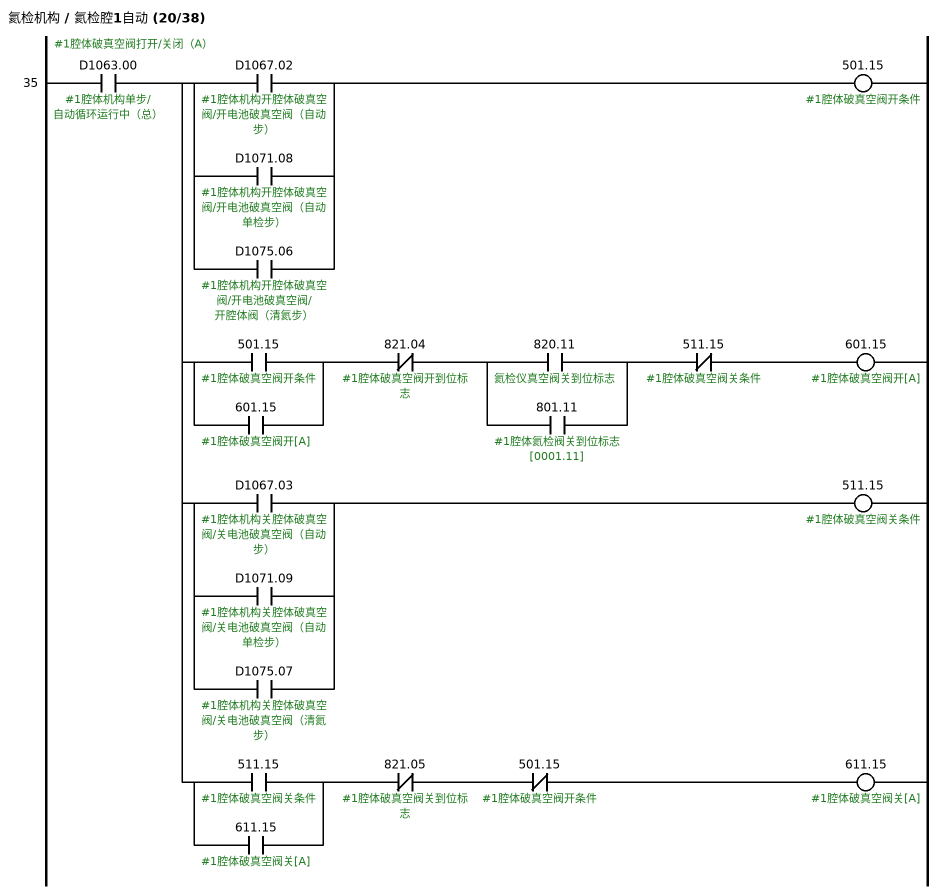
; [picture p216: 氦检机构 / 氦检腔1自动, rungs 35-35]
; rung 35: #1腔体破真空阀打开/关闭（A）
LD D1063.00  ; #1腔体机构单步/自动循环运行中（总）
OUT TR0
LD D1067.02  ; #1腔体机构开腔体破真空阀/开电池破真空阀（自动步）
OR D1071.08  ; #1腔体机构开腔体破真空阀/开电池破真空阀（自动单检步）
OR D1075.06  ; #1腔体机构开腔体破真空阀/开电池破真空阀/开腔体阀（清氦步）
ANDLD
OUT 501.15  ; #1腔体破真空阀开条件
LD TR0
LD 501.15  ; #1腔体破真空阀开条件
OR 601.15  ; #1腔体破真空阀开[A]
ANDLD
ANDNOT 821.04  ; #1腔体破真空阀开到位标志
LD 820.11  ; 氦检仪真空阀关到位标志
OR 801.11  ; #1腔体氦检阀关到位标志[0001.11]
ANDLD
ANDNOT 511.15  ; #1腔体破真空阀关条件
OUT 601.15  ; #1腔体破真空阀开[A]
LD TR0
LD D1067.03  ; #1腔体机构关腔体破真空阀/关电池破真空阀（自动步）
OR D1071.09  ; #1腔体机构关腔体破真空阀/关电池破真空阀（自动单检步）
OR D1075.07  ; #1腔体机构关腔体破真空阀/关电池破真空阀（清氦步）
ANDLD
OUT 511.15  ; #1腔体破真空阀关条件
LD TR0
LD 511.15  ; #1腔体破真空阀关条件
OR 611.15  ; #1腔体破真空阀关[A]
ANDLD
ANDNOT 821.05  ; #1腔体破真空阀关到位标志
ANDNOT 501.15  ; #1腔体破真空阀开条件
OUT 611.15  ; #1腔体破真空阀关[A]

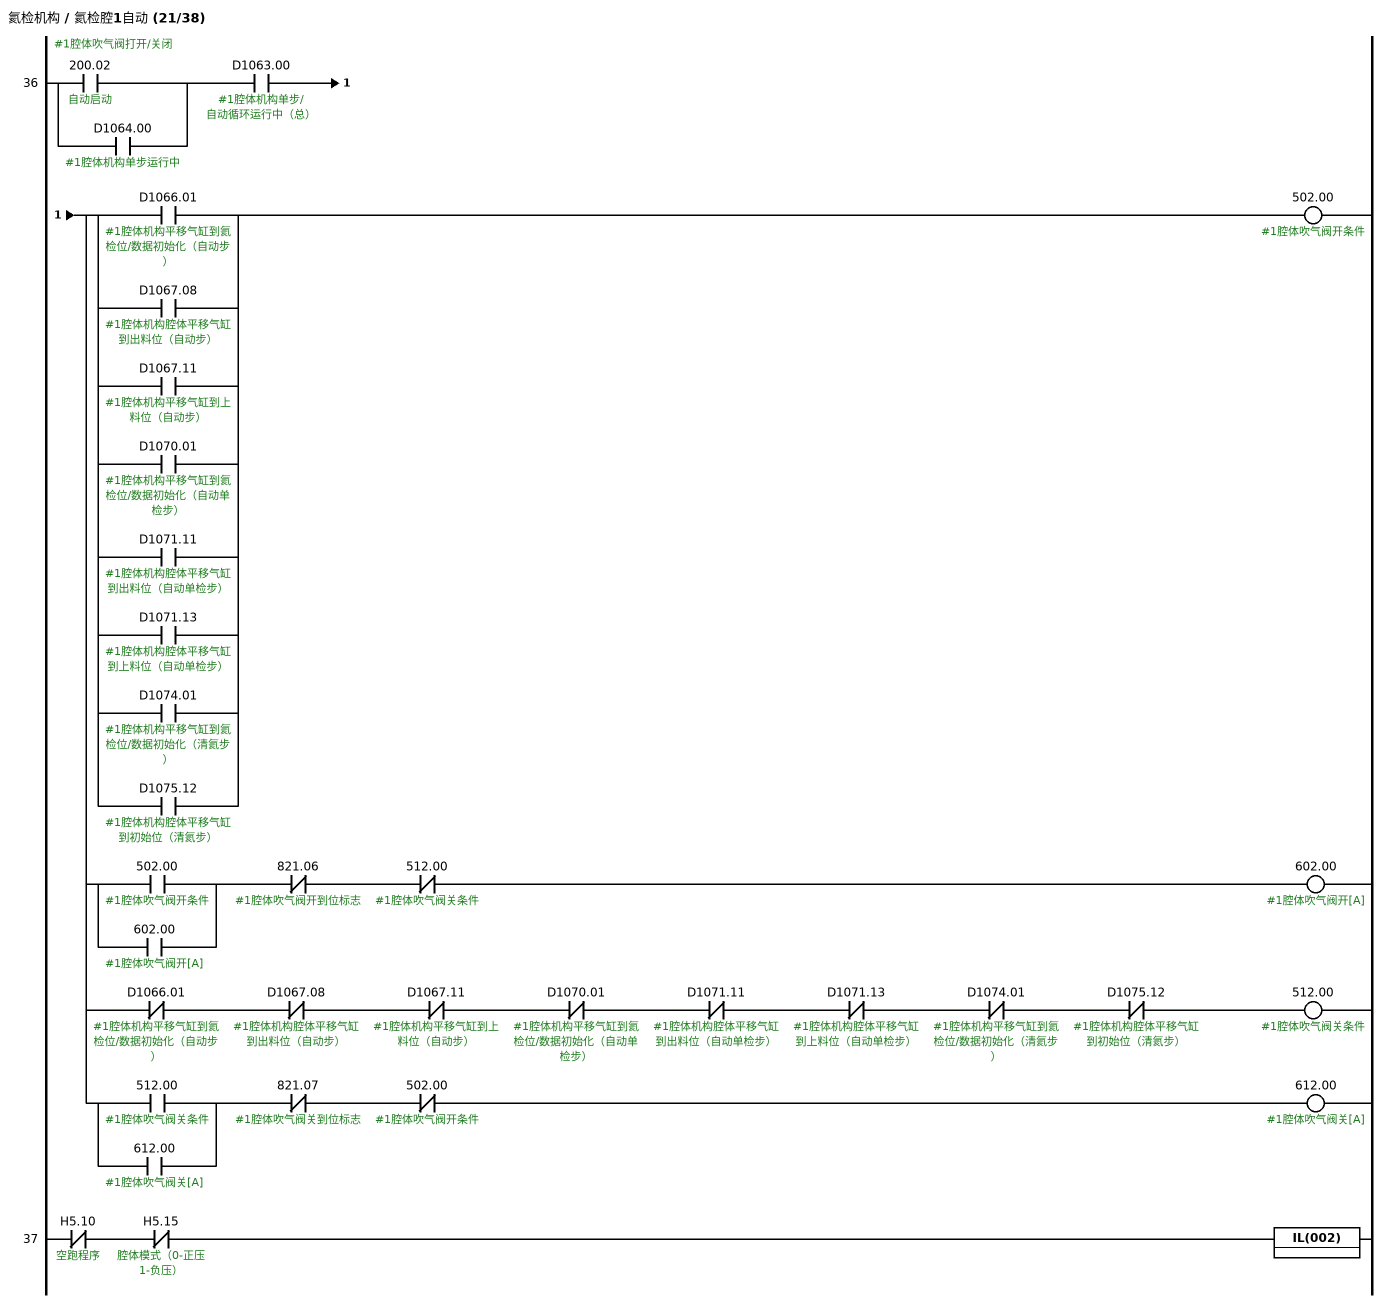
; rung 36: #1腔体吹气阀打开/关闭
LD 200.02  ; 自动启动
OR D1064.00  ; #1腔体机构单步运行中
AND D1063.00  ; #1腔体机构单步/自动循环运行中（总）
OUT TR0
LD D1066.01  ; #1腔体机构平移气缸到氦检位/数据初始化（自动步）
OR D1067.08  ; #1腔体机构腔体平移气缸到出料位（自动步）
OR D1067.11  ; #1腔体机构平移气缸到上料位（自动步）
OR D1070.01  ; #1腔体机构平移气缸到氦检位/数据初始化（自动单检步）
OR D1071.11  ; #1腔体机构腔体平移气缸到出料位（自动单检步）
OR D1071.13  ; #1腔体机构腔体平移气缸到上料位（自动单检步）
OR D1074.01  ; #1腔体机构平移气缸到氦检位/数据初始化（清氦步）
OR D1075.12  ; #1腔体机构腔体平移气缸到初始位（清氦步）
ANDLD
OUT 502.00  ; #1腔体吹气阀开条件
LD TR0
LD 502.00  ; #1腔体吹气阀开条件
OR 602.00  ; #1腔体吹气阀开[A]
ANDLD
ANDNOT 821.06  ; #1腔体吹气阀开到位标志
ANDNOT 512.00  ; #1腔体吹气阀关条件
OUT 602.00  ; #1腔体吹气阀开[A]
LD TR0
ANDNOT D1066.01  ; #1腔体机构平移气缸到氦检位/数据初始化（自动步）
ANDNOT D1067.08  ; #1腔体机构腔体平移气缸到出料位（自动步）
ANDNOT D1067.11  ; #1腔体机构平移气缸到上料位（自动步）
ANDNOT D1070.01  ; #1腔体机构平移气缸到氦检位/数据初始化（自动单检步）
ANDNOT D1071.11  ; #1腔体机构腔体平移气缸到出料位（自动单检步）
ANDNOT D1071.13  ; #1腔体机构腔体平移气缸到上料位（自动单检步）
ANDNOT D1074.01  ; #1腔体机构平移气缸到氦检位/数据初始化（清氦步）
ANDNOT D1075.12  ; #1腔体机构腔体平移气缸到初始位（清氦步）
OUT 512.00  ; #1腔体吹气阀关条件
LD TR0
LD 512.00  ; #1腔体吹气阀关条件
OR 612.00  ; #1腔体吹气阀关[A]
ANDLD
ANDNOT 821.07  ; #1腔体吹气阀关到位标志
ANDNOT 502.00  ; #1腔体吹气阀开条件
OUT 612.00  ; #1腔体吹气阀关[A]
; rung 37
LDNOT H5.10  ; 空跑程序
ANDNOT H5.15  ; 腔体模式（0-正压 1-负压）
IL(002)

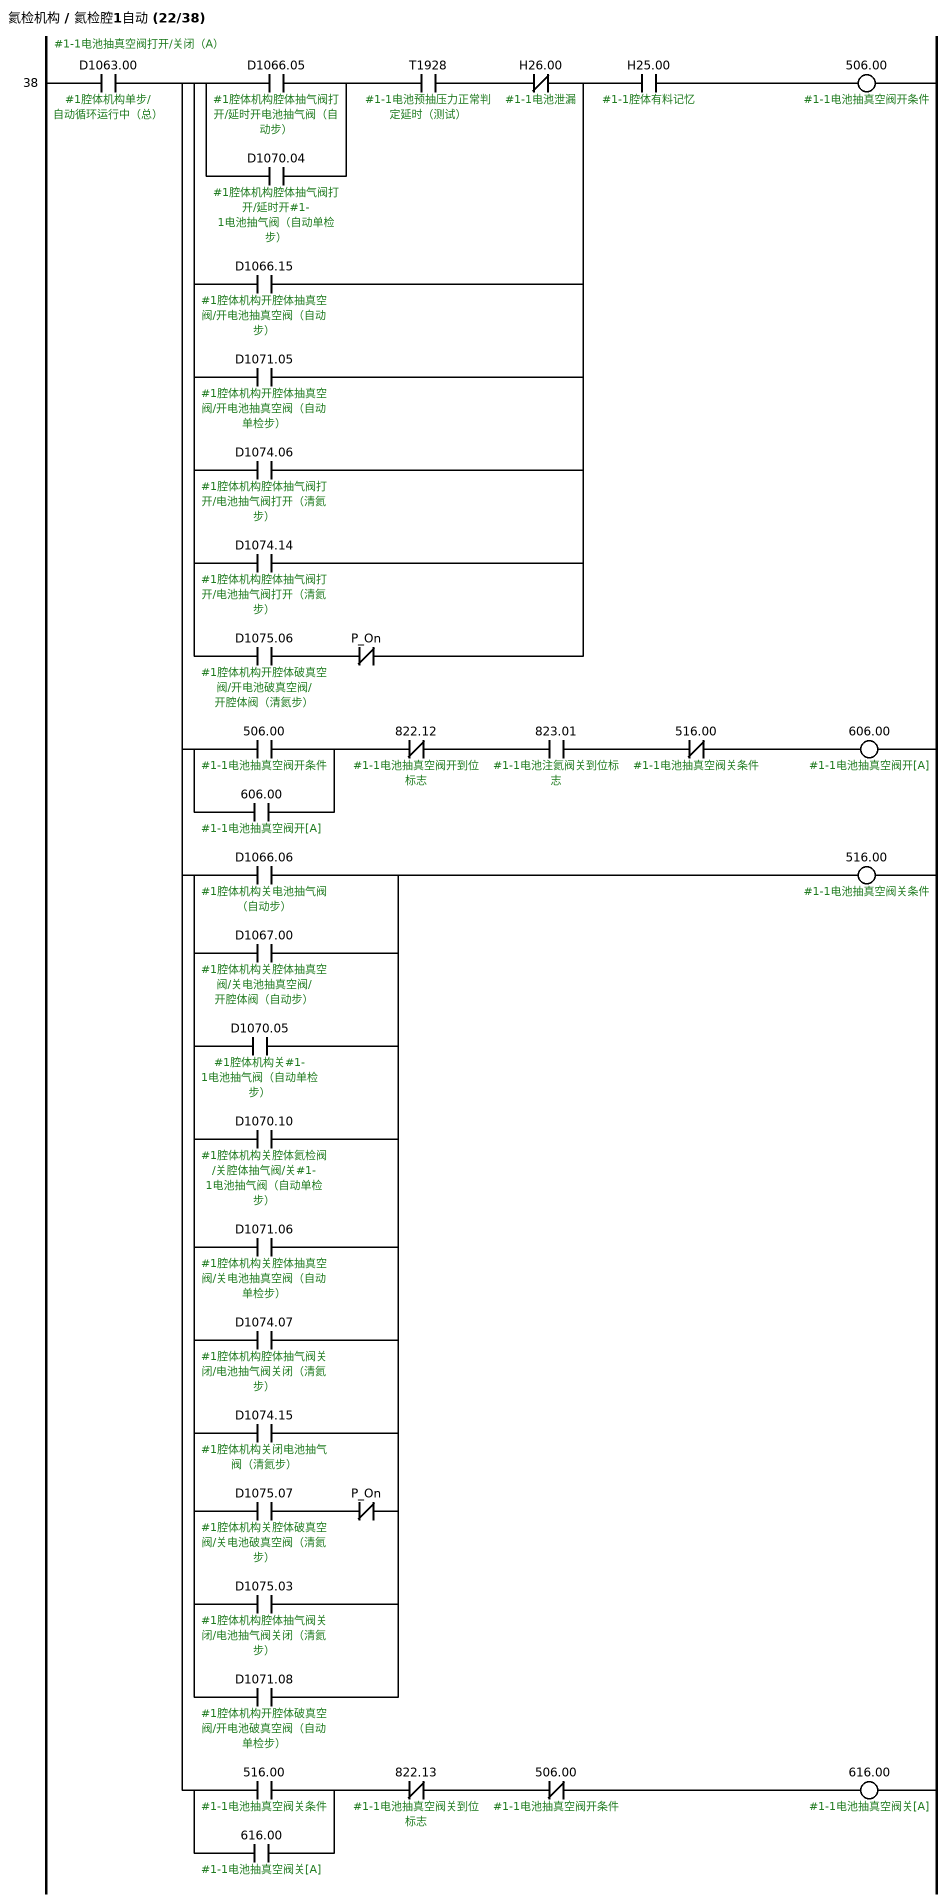
; rung 38: #1-1电池抽真空阀打开/关闭（A）
LD D1063.00  ; #1腔体机构单步/自动循环运行中（总）
OUT TR0
LD D1066.05  ; #1腔体机构腔体抽气阀打开/延时开电池抽气阀（自动步）
OR D1070.04  ; #1腔体机构腔体抽气阀打开/延时开#1-1电池抽气阀（自动单检步）
AND T1928  ; #1-1电池预抽压力正常判定延时（测试）
ANDNOT H26.00  ; #1-1电池泄漏
OR D1066.15  ; #1腔体机构开腔体抽真空阀/开电池抽真空阀（自动步）
OR D1071.05  ; #1腔体机构开腔体抽真空阀/开电池抽真空阀（自动单检步）
OR D1074.06  ; #1腔体机构腔体抽气阀打开/电池抽气阀打开（清氦步）
OR D1074.14  ; #1腔体机构腔体抽气阀打开/电池抽气阀打开（清氦步）
LD D1075.06  ; #1腔体机构开腔体破真空阀/开电池破真空阀/开腔体阀（清氦步）
ANDNOT P_On
ORLD
ANDLD
AND H25.00  ; #1-1腔体有料记忆
OUT 506.00  ; #1-1电池抽真空阀开条件
LD TR0
LD 506.00  ; #1-1电池抽真空阀开条件
OR 606.00  ; #1-1电池抽真空阀开[A]
ANDLD
ANDNOT 822.12  ; #1-1电池抽真空阀开到位标志
AND 823.01  ; #1-1电池注氦阀关到位标志
ANDNOT 516.00  ; #1-1电池抽真空阀关条件
OUT 606.00  ; #1-1电池抽真空阀开[A]
LD TR0
LD D1066.06  ; #1腔体机构关电池抽气阀（自动步）
OR D1067.00  ; #1腔体机构关腔体抽真空阀/关电池抽真空阀/开腔体阀（自动步）
OR D1070.05  ; #1腔体机构关#1-1电池抽气阀（自动单检步）
OR D1070.10  ; #1腔体机构关腔体氦检阀/关腔体抽气阀/关#1-1电池抽气阀（自动单检步）
OR D1071.06  ; #1腔体机构关腔体抽真空阀/关电池抽真空阀（自动单检步）
OR D1074.07  ; #1腔体机构腔体抽气阀关闭/电池抽气阀关闭（清氦步）
OR D1074.15  ; #1腔体机构关闭电池抽气阀（清氦步）
LD D1075.07  ; #1腔体机构关腔体破真空阀/关电池破真空阀（清氦步）
ANDNOT P_On
ORLD
OR D1075.03  ; #1腔体机构腔体抽气阀关闭/电池抽气阀关闭（清氦步）
OR D1071.08  ; #1腔体机构开腔体破真空阀/开电池破真空阀（自动单检步）
ANDLD
OUT 516.00  ; #1-1电池抽真空阀关条件
LD TR0
LD 516.00  ; #1-1电池抽真空阀关条件
OR 616.00  ; #1-1电池抽真空阀关[A]
ANDLD
ANDNOT 822.13  ; #1-1电池抽真空阀关到位标志
ANDNOT 506.00  ; #1-1电池抽真空阀开条件
OUT 616.00  ; #1-1电池抽真空阀关[A]

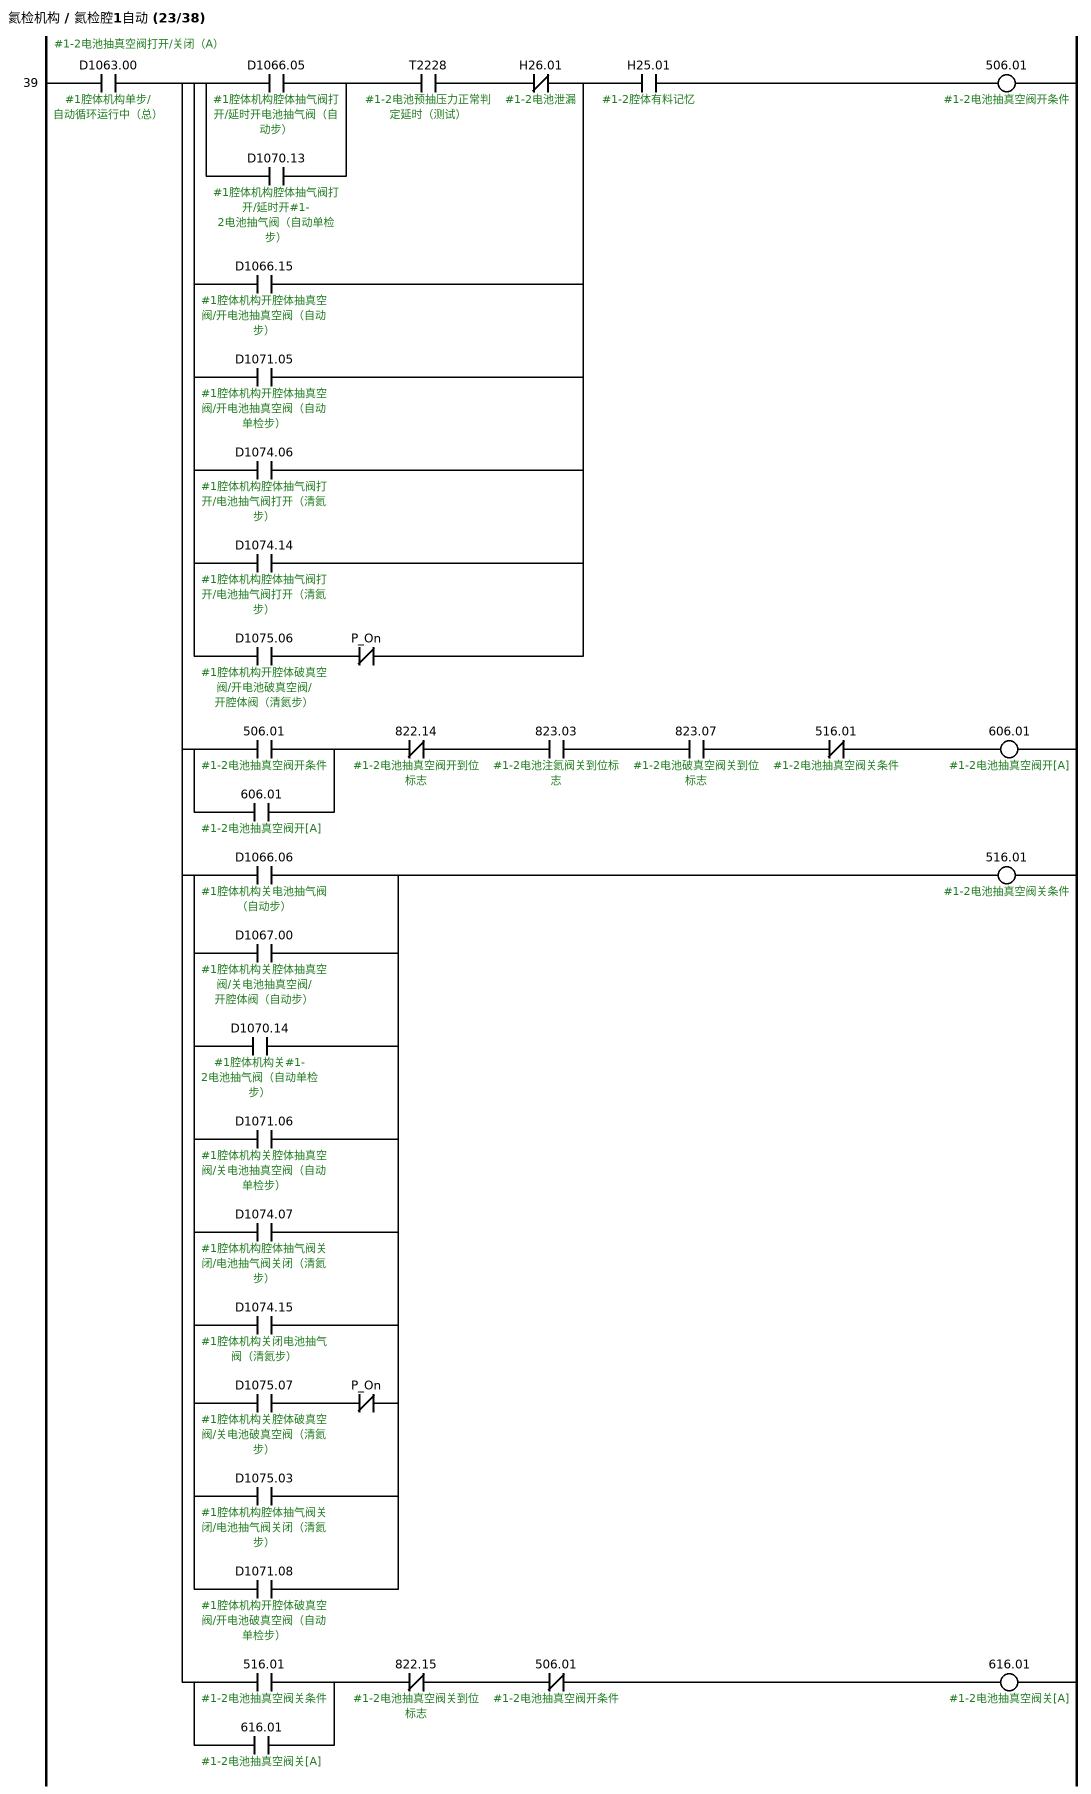
; rung 39: #1-2电池抽真空阀打开/关闭（A）
LD D1063.00  ; #1腔体机构单步/自动循环运行中（总）
OUT TR0
LD D1066.05  ; #1腔体机构腔体抽气阀打开/延时开电池抽气阀（自动步）
OR D1070.13  ; #1腔体机构腔体抽气阀打开/延时开#1-2电池抽气阀（自动单检步）
AND T2228  ; #1-2电池预抽压力正常判定延时（测试）
ANDNOT H26.01  ; #1-2电池泄漏
OR D1066.15  ; #1腔体机构开腔体抽真空阀/开电池抽真空阀（自动步）
OR D1071.05  ; #1腔体机构开腔体抽真空阀/开电池抽真空阀（自动单检步）
OR D1074.06  ; #1腔体机构腔体抽气阀打开/电池抽气阀打开（清氦步）
OR D1074.14  ; #1腔体机构腔体抽气阀打开/电池抽气阀打开（清氦步）
LD D1075.06  ; #1腔体机构开腔体破真空阀/开电池破真空阀/开腔体阀（清氦步）
ANDNOT P_On
ORLD
ANDLD
AND H25.01  ; #1-2腔体有料记忆
OUT 506.01  ; #1-2电池抽真空阀开条件
LD TR0
LD 506.01  ; #1-2电池抽真空阀开条件
OR 606.01  ; #1-2电池抽真空阀开[A]
ANDLD
ANDNOT 822.14  ; #1-2电池抽真空阀开到位标志
AND 823.03  ; #1-2电池注氦阀关到位标志
AND 823.07  ; #1-2电池破真空阀关到位标志
ANDNOT 516.01  ; #1-2电池抽真空阀关条件
OUT 606.01  ; #1-2电池抽真空阀开[A]
LD TR0
LD D1066.06  ; #1腔体机构关电池抽气阀（自动步）
OR D1067.00  ; #1腔体机构关腔体抽真空阀/关电池抽真空阀/开腔体阀（自动步）
OR D1070.14  ; #1腔体机构关#1-2电池抽气阀（自动单检步）
OR D1071.06  ; #1腔体机构关腔体抽真空阀/关电池抽真空阀（自动单检步）
OR D1074.07  ; #1腔体机构腔体抽气阀关闭/电池抽气阀关闭（清氦步）
OR D1074.15  ; #1腔体机构关闭电池抽气阀（清氦步）
LD D1075.07  ; #1腔体机构关腔体破真空阀/关电池破真空阀（清氦步）
ANDNOT P_On
ORLD
OR D1075.03  ; #1腔体机构腔体抽气阀关闭/电池抽气阀关闭（清氦步）
OR D1071.08  ; #1腔体机构开腔体破真空阀/开电池破真空阀（自动单检步）
ANDLD
OUT 516.01  ; #1-2电池抽真空阀关条件
LD TR0
LD 516.01  ; #1-2电池抽真空阀关条件
OR 616.01  ; #1-2电池抽真空阀关[A]
ANDLD
ANDNOT 822.15  ; #1-2电池抽真空阀关到位标志
ANDNOT 506.01  ; #1-2电池抽真空阀开条件
OUT 616.01  ; #1-2电池抽真空阀关[A]

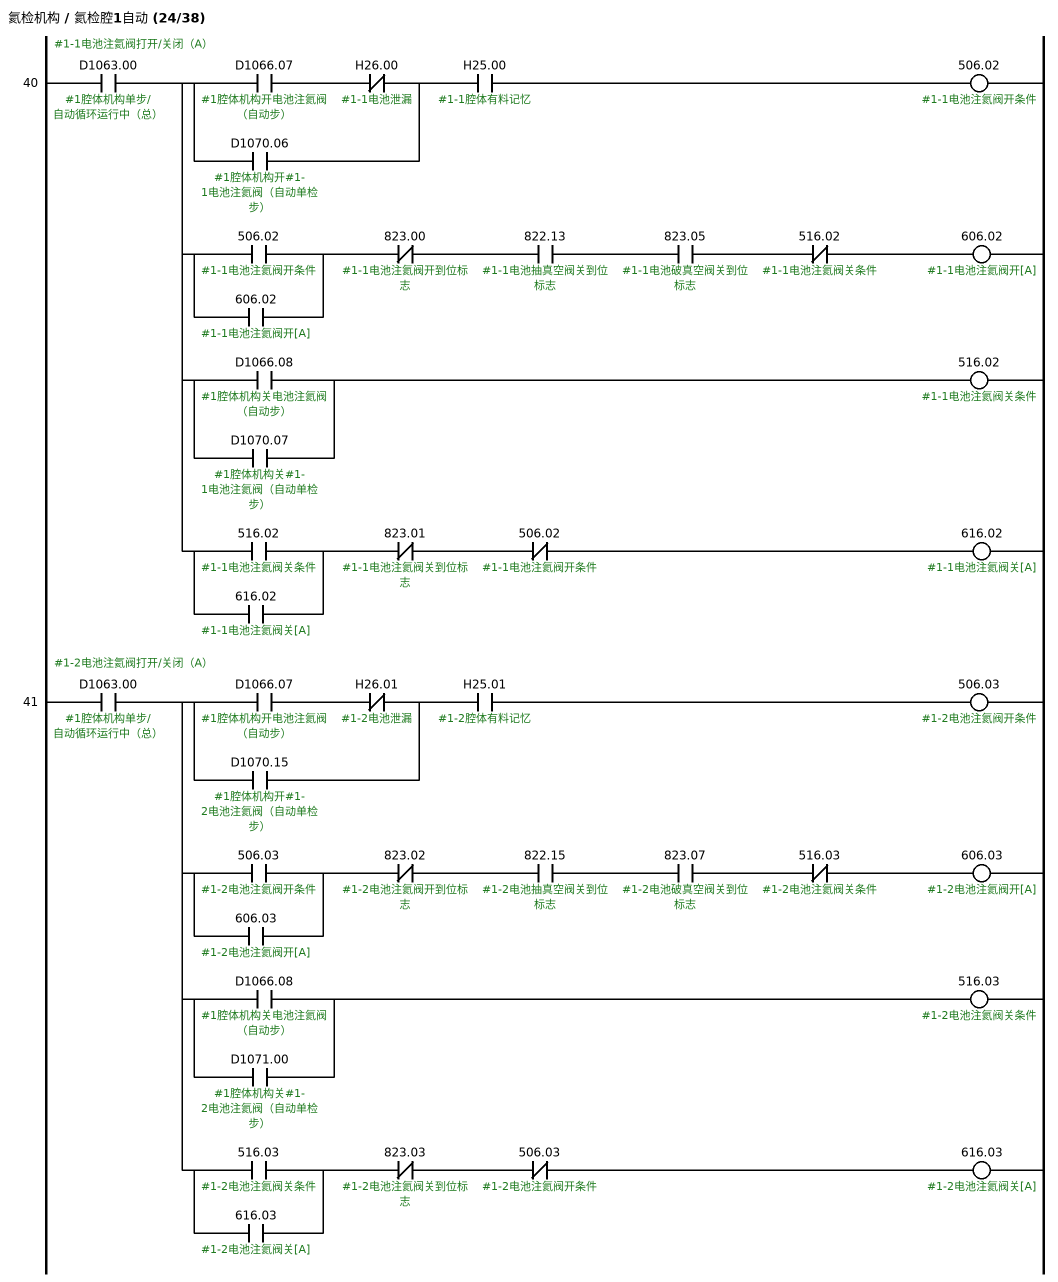
; rung 40: #1-1电池注氦阀打开/关闭（A）
LD D1063.00  ; #1腔体机构单步/自动循环运行中（总）
OUT TR0
LD D1066.07  ; #1腔体机构开电池注氦阀（自动步）
ANDNOT H26.00  ; #1-1电池泄漏
OR D1070.06  ; #1腔体机构开#1-1电池注氦阀（自动单检步）
ANDLD
AND H25.00  ; #1-1腔体有料记忆
OUT 506.02  ; #1-1电池注氦阀开条件
LD TR0
LD 506.02  ; #1-1电池注氦阀开条件
OR 606.02  ; #1-1电池注氦阀开[A]
ANDLD
ANDNOT 823.00  ; #1-1电池注氦阀开到位标志
AND 822.13  ; #1-1电池抽真空阀关到位标志
AND 823.05  ; #1-1电池破真空阀关到位标志
ANDNOT 516.02  ; #1-1电池注氦阀关条件
OUT 606.02  ; #1-1电池注氦阀开[A]
LD TR0
LD D1066.08  ; #1腔体机构关电池注氦阀（自动步）
OR D1070.07  ; #1腔体机构关#1-1电池注氦阀（自动单检步）
ANDLD
OUT 516.02  ; #1-1电池注氦阀关条件
LD TR0
LD 516.02  ; #1-1电池注氦阀关条件
OR 616.02  ; #1-1电池注氦阀关[A]
ANDLD
ANDNOT 823.01  ; #1-1电池注氦阀关到位标志
ANDNOT 506.02  ; #1-1电池注氦阀开条件
OUT 616.02  ; #1-1电池注氦阀关[A]
; rung 41: #1-2电池注氦阀打开/关闭（A）
LD D1063.00  ; #1腔体机构单步/自动循环运行中（总）
OUT TR0
LD D1066.07  ; #1腔体机构开电池注氦阀（自动步）
ANDNOT H26.01  ; #1-2电池泄漏
OR D1070.15  ; #1腔体机构开#1-2电池注氦阀（自动单检步）
ANDLD
AND H25.01  ; #1-2腔体有料记忆
OUT 506.03  ; #1-2电池注氦阀开条件
LD TR0
LD 506.03  ; #1-2电池注氦阀开条件
OR 606.03  ; #1-2电池注氦阀开[A]
ANDLD
ANDNOT 823.02  ; #1-2电池注氦阀开到位标志
AND 822.15  ; #1-2电池抽真空阀关到位标志
AND 823.07  ; #1-2电池破真空阀关到位标志
ANDNOT 516.03  ; #1-2电池注氦阀关条件
OUT 606.03  ; #1-2电池注氦阀开[A]
LD TR0
LD D1066.08  ; #1腔体机构关电池注氦阀（自动步）
OR D1071.00  ; #1腔体机构关#1-2电池注氦阀（自动单检步）
ANDLD
OUT 516.03  ; #1-2电池注氦阀关条件
LD TR0
LD 516.03  ; #1-2电池注氦阀关条件
OR 616.03  ; #1-2电池注氦阀关[A]
ANDLD
ANDNOT 823.03  ; #1-2电池注氦阀关到位标志
ANDNOT 506.03  ; #1-2电池注氦阀开条件
OUT 616.03  ; #1-2电池注氦阀关[A]

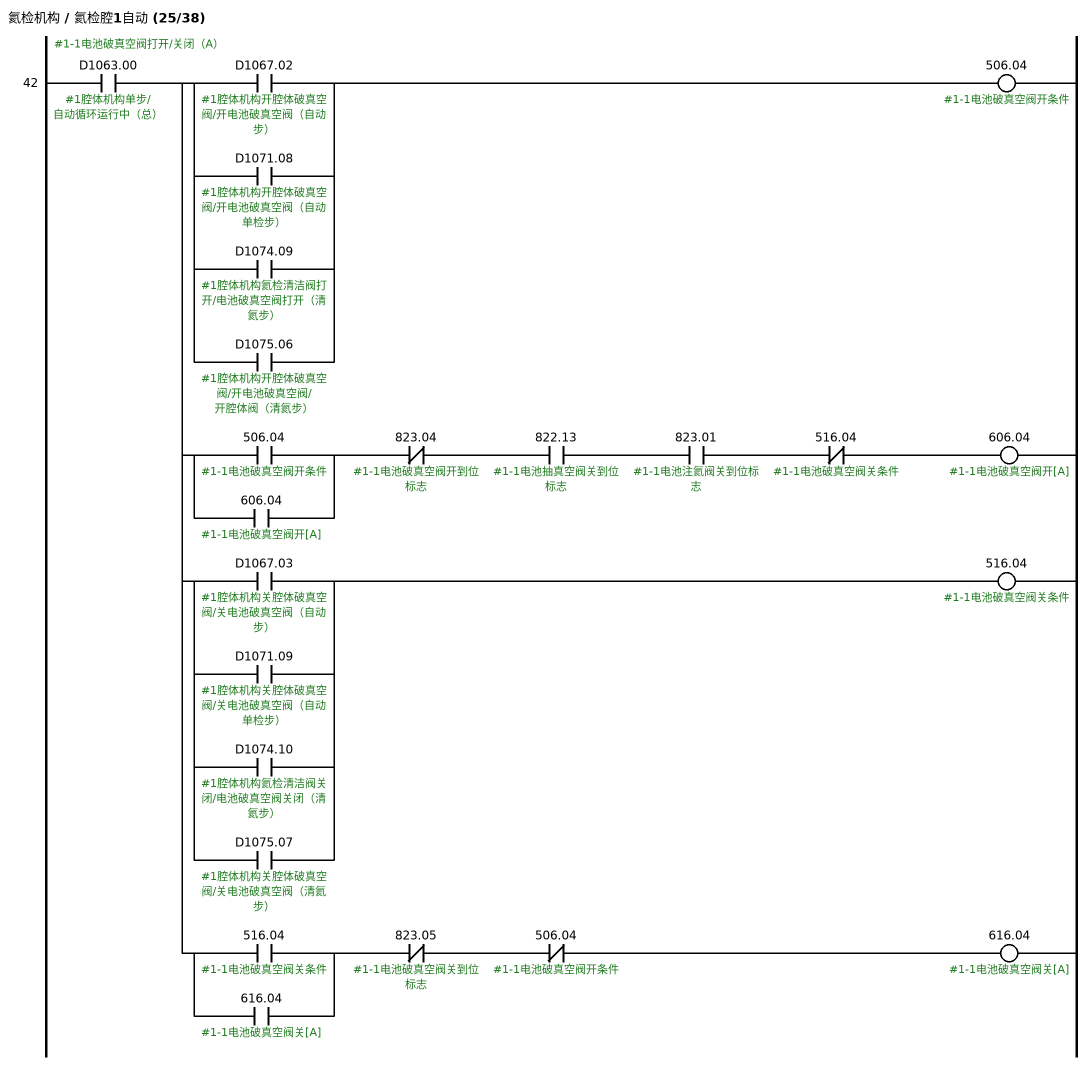
; rung 42: #1-1电池破真空阀打开/关闭（A）
LD D1063.00  ; #1腔体机构单步/自动循环运行中（总）
OUT TR0
LD D1067.02  ; #1腔体机构开腔体破真空阀/开电池破真空阀（自动步）
OR D1071.08  ; #1腔体机构开腔体破真空阀/开电池破真空阀（自动单检步）
OR D1074.09  ; #1腔体机构氦检清洁阀打开/电池破真空阀打开（清氦步）
OR D1075.06  ; #1腔体机构开腔体破真空阀/开电池破真空阀/开腔体阀（清氦步）
ANDLD
OUT 506.04  ; #1-1电池破真空阀开条件
LD TR0
LD 506.04  ; #1-1电池破真空阀开条件
OR 606.04  ; #1-1电池破真空阀开[A]
ANDLD
ANDNOT 823.04  ; #1-1电池破真空阀开到位标志
AND 822.13  ; #1-1电池抽真空阀关到位标志
AND 823.01  ; #1-1电池注氦阀关到位标志
ANDNOT 516.04  ; #1-1电池破真空阀关条件
OUT 606.04  ; #1-1电池破真空阀开[A]
LD TR0
LD D1067.03  ; #1腔体机构关腔体破真空阀/关电池破真空阀（自动步）
OR D1071.09  ; #1腔体机构关腔体破真空阀/关电池破真空阀（自动单检步）
OR D1074.10  ; #1腔体机构氦检清洁阀关闭/电池破真空阀关闭（清氦步）
OR D1075.07  ; #1腔体机构关腔体破真空阀/关电池破真空阀（清氦步）
ANDLD
OUT 516.04  ; #1-1电池破真空阀关条件
LD TR0
LD 516.04  ; #1-1电池破真空阀关条件
OR 616.04  ; #1-1电池破真空阀关[A]
ANDLD
ANDNOT 823.05  ; #1-1电池破真空阀关到位标志
ANDNOT 506.04  ; #1-1电池破真空阀开条件
OUT 616.04  ; #1-1电池破真空阀关[A]

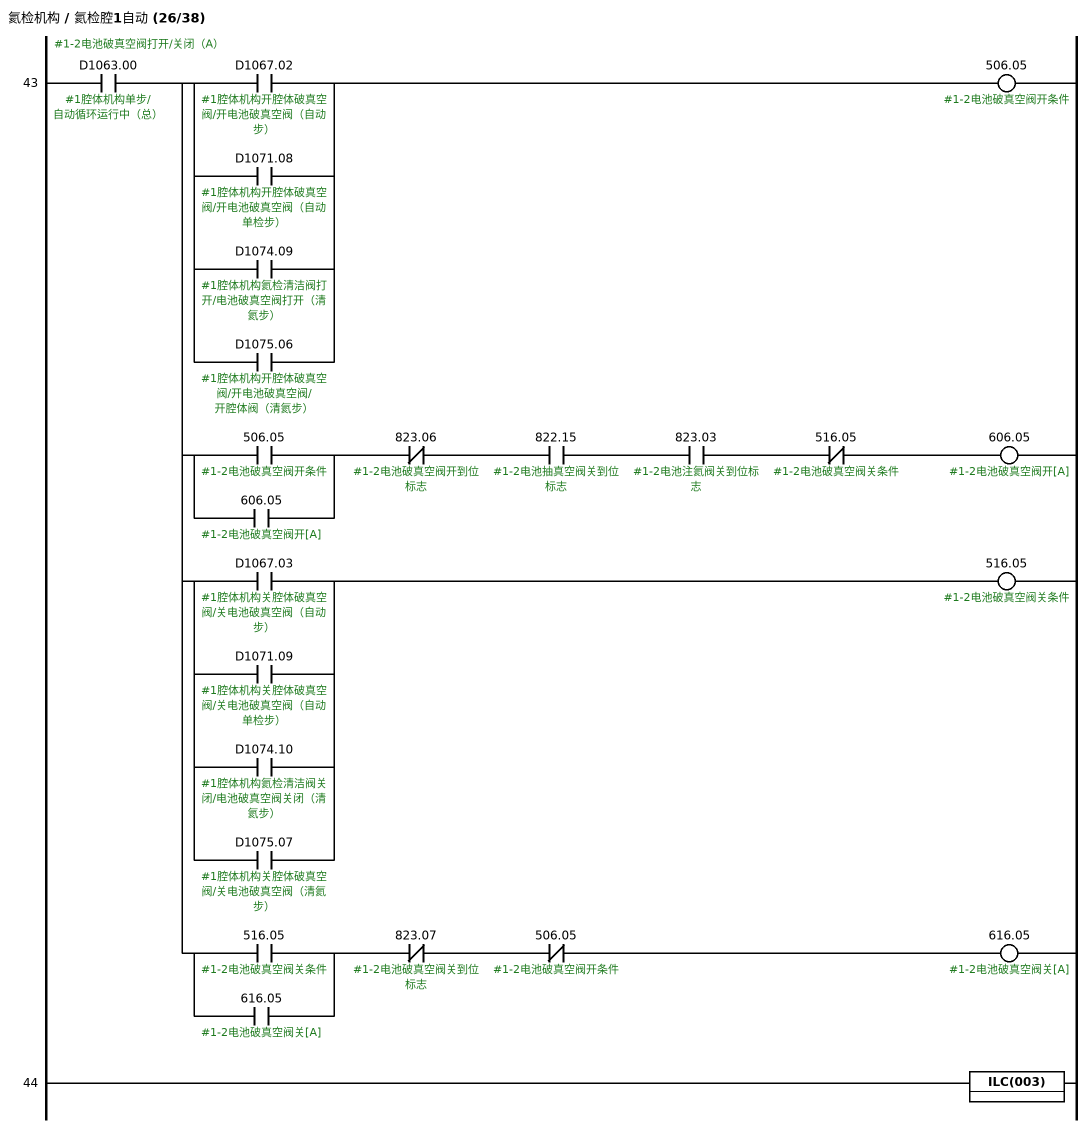
; rung 43: #1-2电池破真空阀打开/关闭（A）
LD D1063.00  ; #1腔体机构单步/自动循环运行中（总）
OUT TR0
LD D1067.02  ; #1腔体机构开腔体破真空阀/开电池破真空阀（自动步）
OR D1071.08  ; #1腔体机构开腔体破真空阀/开电池破真空阀（自动单检步）
OR D1074.09  ; #1腔体机构氦检清洁阀打开/电池破真空阀打开（清氦步）
OR D1075.06  ; #1腔体机构开腔体破真空阀/开电池破真空阀/开腔体阀（清氦步）
ANDLD
OUT 506.05  ; #1-2电池破真空阀开条件
LD TR0
LD 506.05  ; #1-2电池破真空阀开条件
OR 606.05  ; #1-2电池破真空阀开[A]
ANDLD
ANDNOT 823.06  ; #1-2电池破真空阀开到位标志
AND 822.15  ; #1-2电池抽真空阀关到位标志
AND 823.03  ; #1-2电池注氦阀关到位标志
ANDNOT 516.05  ; #1-2电池破真空阀关条件
OUT 606.05  ; #1-2电池破真空阀开[A]
LD TR0
LD D1067.03  ; #1腔体机构关腔体破真空阀/关电池破真空阀（自动步）
OR D1071.09  ; #1腔体机构关腔体破真空阀/关电池破真空阀（自动单检步）
OR D1074.10  ; #1腔体机构氦检清洁阀关闭/电池破真空阀关闭（清氦步）
OR D1075.07  ; #1腔体机构关腔体破真空阀/关电池破真空阀（清氦步）
ANDLD
OUT 516.05  ; #1-2电池破真空阀关条件
LD TR0
LD 516.05  ; #1-2电池破真空阀关条件
OR 616.05  ; #1-2电池破真空阀关[A]
ANDLD
ANDNOT 823.07  ; #1-2电池破真空阀关到位标志
ANDNOT 506.05  ; #1-2电池破真空阀开条件
OUT 616.05  ; #1-2电池破真空阀关[A]
; rung 44
ILC(003)

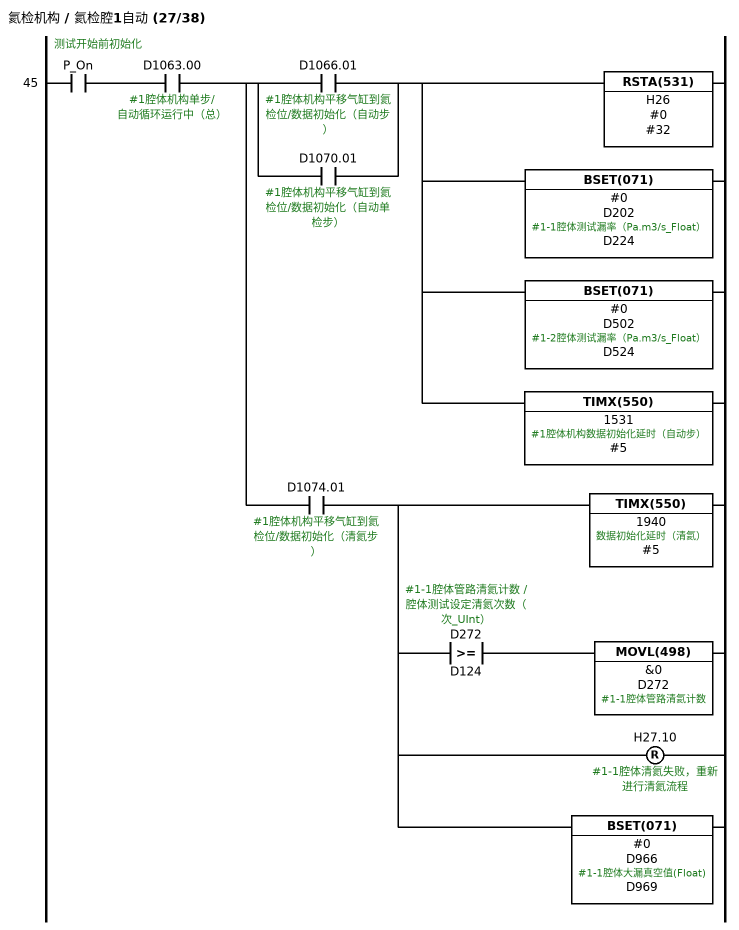
; rung 45: 测试开始前初始化
LD P_On
AND D1063.00  ; #1腔体机构单步/自动循环运行中（总）
OUT TR0
LD D1066.01  ; #1腔体机构平移气缸到氦检位/数据初始化（自动步）
OR D1070.01  ; #1腔体机构平移气缸到氦检位/数据初始化（自动单检步）
ANDLD
RSTA(531) H26 #0 #32
BSET(071) #0 D202 D224  ; #1-1腔体测试漏率（Pa.m3/s_Float）
BSET(071) #0 D502 D524  ; #1-2腔体测试漏率（Pa.m3/s_Float）
TIMX(550) 1531 #5  ; #1腔体机构数据初始化延时（自动步）
LD TR0
AND D1074.01  ; #1腔体机构平移气缸到氦检位/数据初始化（清氦步）
OUT TR0
TIMX(550) 1940 #5  ; 数据初始化延时（清氦）
AND>=(325) D272 D124  ; #1-1腔体管路清氦计数, 腔体测试设定清氦次数（次_UInt）
MOVL(498) &0 D272  ; #1-1腔体管路清氦计数
LD TR0
RSET H27.10  ; #1-1腔体清氦失败，重新进行清氦流程
BSET(071) #0 D966 D969  ; #1-1腔体大漏真空值(Float)

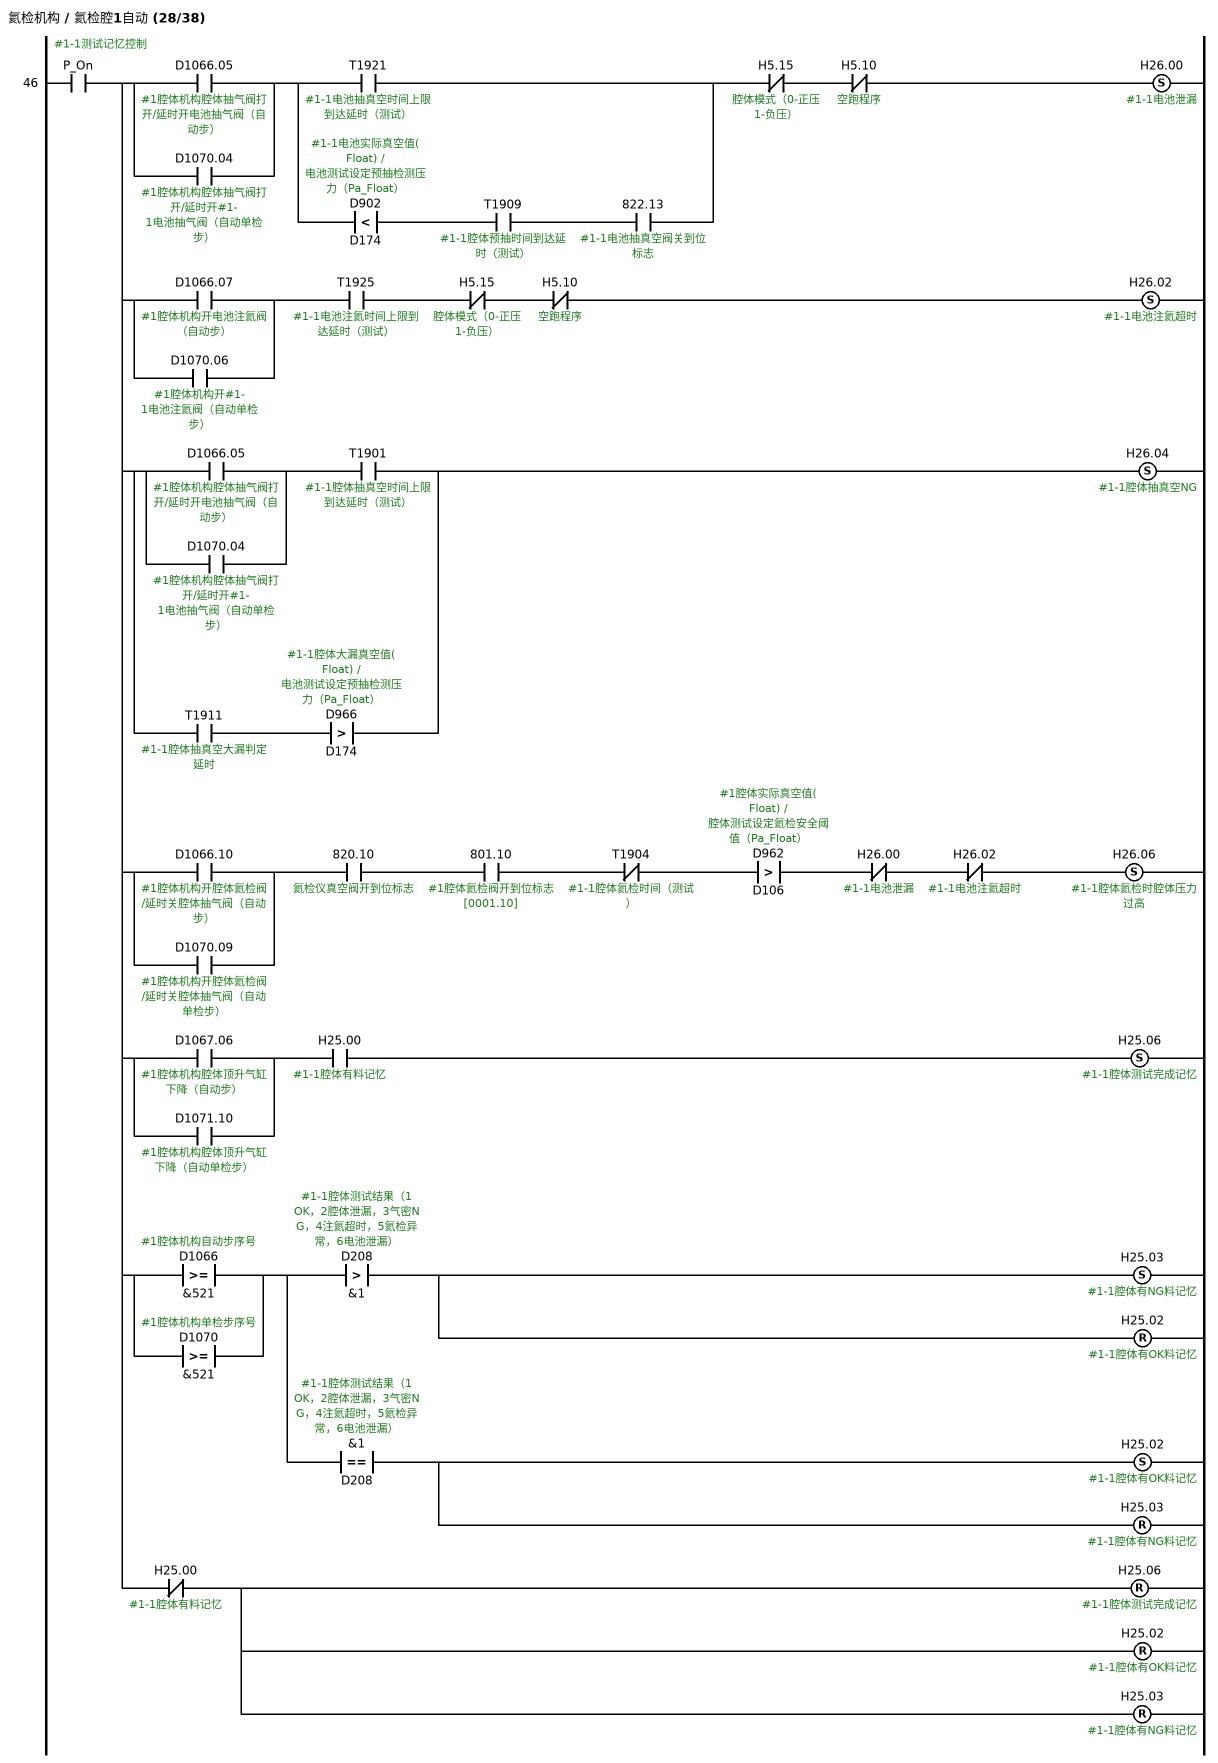
; rung 46: #1-1测试记忆控制
LD P_On
OUT TR0
LD D1066.05  ; #1腔体机构腔体抽气阀打开/延时开电池抽气阀（自动步）
OR D1070.04  ; #1腔体机构腔体抽气阀打开/延时开#1-1电池抽气阀（自动单检步）
ANDLD
LD T1921  ; #1-1电池抽真空时间上限到达延时（测试）
LD<F(331) D902 D174  ; #1-1电池实际真空值(Float), 电池测试设定预抽检测压力（Pa_Float）
AND T1909  ; #1-1腔体预抽时间到达延时（测试）
AND 822.13  ; #1-1电池抽真空阀关到位标志
ORLD
ANDLD
ANDNOT H5.15  ; 腔体模式（0-正压 1-负压）
ANDNOT H5.10  ; 空跑程序
SET H26.00  ; #1-1电池泄漏
LD TR0
LD D1066.07  ; #1腔体机构开电池注氦阀（自动步）
OR D1070.06  ; #1腔体机构开#1-1电池注氦阀（自动单检步）
ANDLD
AND T1925  ; #1-1电池注氦时间上限到达延时（测试）
ANDNOT H5.15  ; 腔体模式（0-正压 1-负压）
ANDNOT H5.10  ; 空跑程序
SET H26.02  ; #1-1电池注氦超时
LD TR0
LD D1066.05  ; #1腔体机构腔体抽气阀打开/延时开电池抽气阀（自动步）
OR D1070.04  ; #1腔体机构腔体抽气阀打开/延时开#1-1电池抽气阀（自动单检步）
AND T1901  ; #1-1腔体抽真空时间上限到达延时（测试）
LD T1911  ; #1-1腔体抽真空大漏判定延时
AND>F(333) D966 D174  ; #1-1腔体大漏真空值(Float), 电池测试设定预抽检测压力（Pa_Float）
ORLD
ANDLD
SET H26.04  ; #1-1腔体抽真空NG
LD TR0
LD D1066.10  ; #1腔体机构开腔体氦检阀/延时关腔体抽气阀（自动步）
OR D1070.09  ; #1腔体机构开腔体氦检阀/延时关腔体抽气阀（自动单检步）
ANDLD
AND 820.10  ; 氦检仪真空阀开到位标志
AND 801.10  ; #1腔体氦检阀开到位标志[0001.10]
ANDNOT T1904  ; #1-1腔体氦检时间（测试）
AND>F(333) D962 D106  ; #1腔体实际真空值(Float), 腔体测试设定氦检安全阈值（Pa_Float）
ANDNOT H26.00  ; #1-1电池泄漏
ANDNOT H26.02  ; #1-1电池注氦超时
SET H26.06  ; #1-1腔体氦检时腔体压力过高
LD TR0
LD D1067.06  ; #1腔体机构腔体顶升气缸下降（自动步）
OR D1071.10  ; #1腔体机构腔体顶升气缸下降（自动单检步）
ANDLD
AND H25.00  ; #1-1腔体有料记忆
SET H25.06  ; #1-1腔体测试完成记忆
LD TR0
LD>=L(326) D1066 &521  ; #1腔体机构自动步序号
OR>=L(326) D1070 &521  ; #1腔体机构单检步序号
ANDLD
OUT TR1
AND>(320) D208 &1  ; #1-1腔体测试结果（1 OK，2腔体泄漏，3气密NG，4注氦超时，5氦检异常，6电池泄漏）
SET H25.03  ; #1-1腔体有NG料记忆
RSET H25.02  ; #1-1腔体有OK料记忆
LD TR1
AND=(300) &1 D208  ; #1-1腔体测试结果（1 OK，2腔体泄漏，3气密NG，4注氦超时，5氦检异常，6电池泄漏）
SET H25.02  ; #1-1腔体有OK料记忆
RSET H25.03  ; #1-1腔体有NG料记忆
LD TR0
ANDNOT H25.00  ; #1-1腔体有料记忆
RSET H25.06  ; #1-1腔体测试完成记忆
RSET H25.02  ; #1-1腔体有OK料记忆
RSET H25.03  ; #1-1腔体有NG料记忆

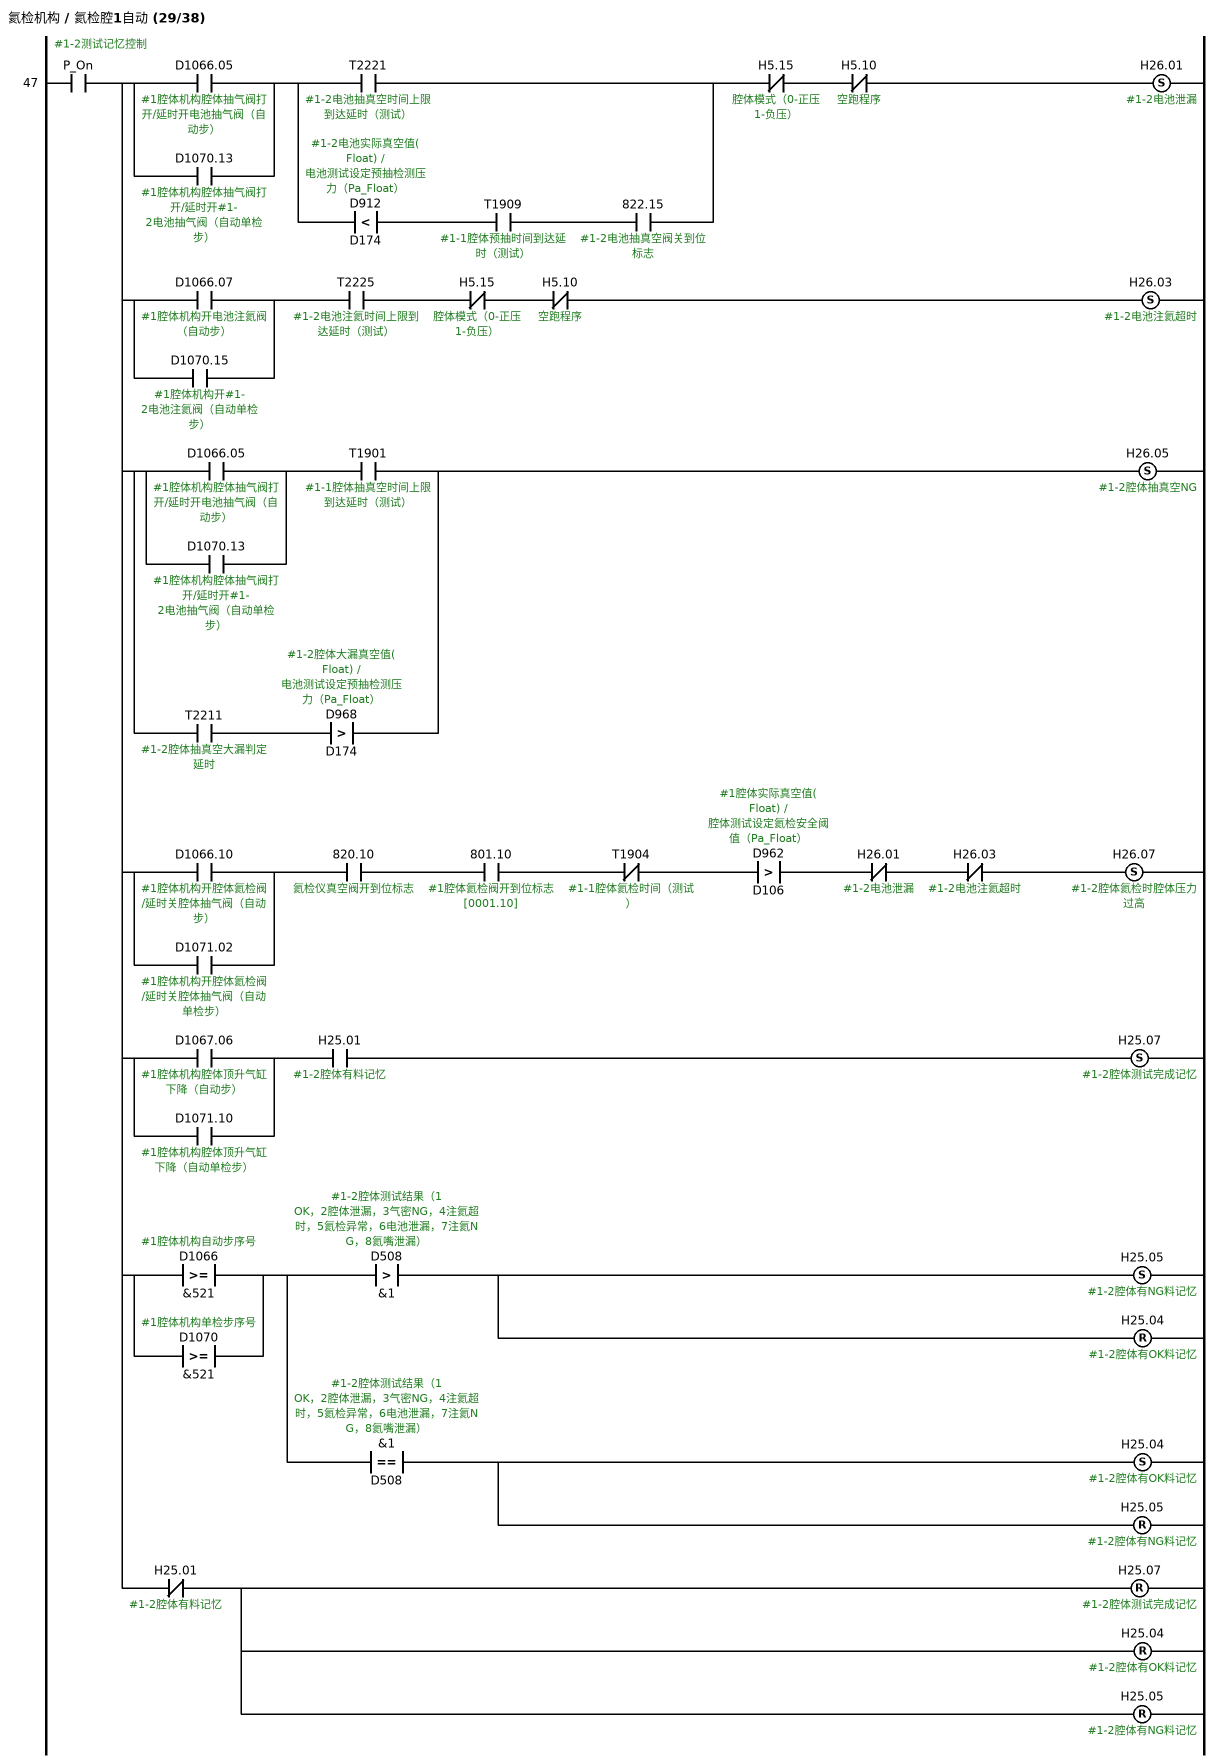
; rung 47: #1-2测试记忆控制
LD P_On
OUT TR0
LD D1066.05  ; #1腔体机构腔体抽气阀打开/延时开电池抽气阀（自动步）
OR D1070.13  ; #1腔体机构腔体抽气阀打开/延时开#1-2电池抽气阀（自动单检步）
ANDLD
LD T2221  ; #1-2电池抽真空时间上限到达延时（测试）
LD<F(331) D912 D174  ; #1-2电池实际真空值(Float), 电池测试设定预抽检测压力（Pa_Float）
AND T1909  ; #1-1腔体预抽时间到达延时（测试）
AND 822.15  ; #1-2电池抽真空阀关到位标志
ORLD
ANDLD
ANDNOT H5.15  ; 腔体模式（0-正压 1-负压）
ANDNOT H5.10  ; 空跑程序
SET H26.01  ; #1-2电池泄漏
LD TR0
LD D1066.07  ; #1腔体机构开电池注氦阀（自动步）
OR D1070.15  ; #1腔体机构开#1-2电池注氦阀（自动单检步）
ANDLD
AND T2225  ; #1-2电池注氦时间上限到达延时（测试）
ANDNOT H5.15  ; 腔体模式（0-正压 1-负压）
ANDNOT H5.10  ; 空跑程序
SET H26.03  ; #1-2电池注氦超时
LD TR0
LD D1066.05  ; #1腔体机构腔体抽气阀打开/延时开电池抽气阀（自动步）
OR D1070.13  ; #1腔体机构腔体抽气阀打开/延时开#1-2电池抽气阀（自动单检步）
AND T1901  ; #1-1腔体抽真空时间上限到达延时（测试）
LD T2211  ; #1-2腔体抽真空大漏判定延时
AND>F(333) D968 D174  ; #1-2腔体大漏真空值(Float), 电池测试设定预抽检测压力（Pa_Float）
ORLD
ANDLD
SET H26.05  ; #1-2腔体抽真空NG
LD TR0
LD D1066.10  ; #1腔体机构开腔体氦检阀/延时关腔体抽气阀（自动步）
OR D1071.02  ; #1腔体机构开腔体氦检阀/延时关腔体抽气阀（自动单检步）
ANDLD
AND 820.10  ; 氦检仪真空阀开到位标志
AND 801.10  ; #1腔体氦检阀开到位标志[0001.10]
ANDNOT T1904  ; #1-1腔体氦检时间（测试）
AND>F(333) D962 D106  ; #1腔体实际真空值(Float), 腔体测试设定氦检安全阈值（Pa_Float）
ANDNOT H26.01  ; #1-2电池泄漏
ANDNOT H26.03  ; #1-2电池注氦超时
SET H26.07  ; #1-2腔体氦检时腔体压力过高
LD TR0
LD D1067.06  ; #1腔体机构腔体顶升气缸下降（自动步）
OR D1071.10  ; #1腔体机构腔体顶升气缸下降（自动单检步）
ANDLD
AND H25.01  ; #1-2腔体有料记忆
SET H25.07  ; #1-2腔体测试完成记忆
LD TR0
LD>=L(326) D1066 &521  ; #1腔体机构自动步序号
OR>=L(326) D1070 &521  ; #1腔体机构单检步序号
ANDLD
OUT TR1
AND>(320) D508 &1  ; #1-2腔体测试结果（1 OK，2腔体泄漏，3气密NG，4注氦超时，5氦检异常，6电池泄漏，7注氦NG，8氦嘴泄漏）
SET H25.05  ; #1-2腔体有NG料记忆
RSET H25.04  ; #1-2腔体有OK料记忆
LD TR1
AND=(300) &1 D508  ; #1-2腔体测试结果（1 OK，2腔体泄漏，3气密NG，4注氦超时，5氦检异常，6电池泄漏，7注氦NG，8氦嘴泄漏）
SET H25.04  ; #1-2腔体有OK料记忆
RSET H25.05  ; #1-2腔体有NG料记忆
LD TR0
ANDNOT H25.01  ; #1-2腔体有料记忆
RSET H25.07  ; #1-2腔体测试完成记忆
RSET H25.04  ; #1-2腔体有OK料记忆
RSET H25.05  ; #1-2腔体有NG料记忆

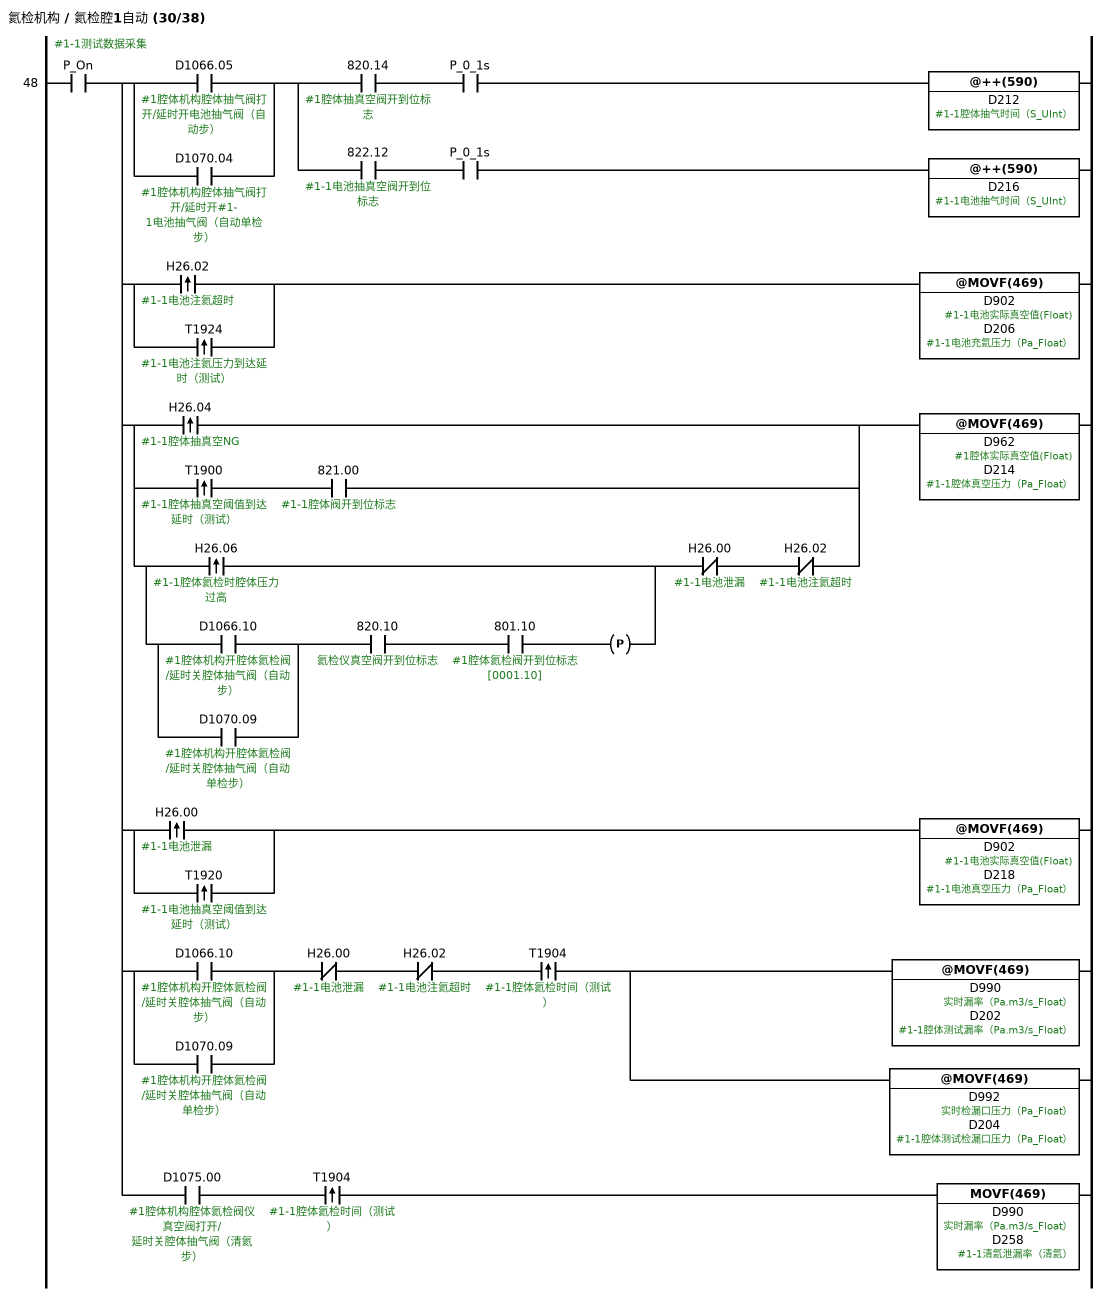
; rung 48: #1-1测试数据采集
LD P_On
OUT TR0
LD D1066.05  ; #1腔体机构腔体抽气阀打开/延时开电池抽气阀（自动步）
OR D1070.04  ; #1腔体机构腔体抽气阀打开/延时开#1-1电池抽气阀（自动单检步）
ANDLD
OUT TR1
AND 820.14  ; #1腔体抽真空阀开到位标志
AND P_0_1s
@++(590) D212  ; #1-1腔体抽气时间（S_UInt）
LD TR1
AND 822.12  ; #1-1电池抽真空阀开到位标志
AND P_0_1s
@++(590) D216  ; #1-1电池抽气时间（S_UInt）
LD TR0
@LD H26.02  ; #1-1电池注氦超时
@OR T1924  ; #1-1电池注氦压力到达延时（测试）
ANDLD
@MOVF(469) D902 D206  ; #1-1电池实际真空值(Float), #1-1电池充氦压力（Pa_Float）
LD TR0
@LD H26.04  ; #1-1腔体抽真空NG
@LD T1900  ; #1-1腔体抽真空阈值到达延时（测试）
AND 821.00  ; #1-1腔体阀开到位标志
ORLD
@LD H26.06  ; #1-1腔体氦检时腔体压力过高
LD D1066.10  ; #1腔体机构开腔体氦检阀/延时关腔体抽气阀（自动步）
OR D1070.09  ; #1腔体机构开腔体氦检阀/延时关腔体抽气阀（自动单检步）
AND 820.10  ; 氦检仪真空阀开到位标志
AND 801.10  ; #1腔体氦检阀开到位标志[0001.10]
UP(521)
ORLD
ANDNOT H26.00  ; #1-1电池泄漏
ANDNOT H26.02  ; #1-1电池注氦超时
ORLD
ANDLD
@MOVF(469) D962 D214  ; #1腔体实际真空值(Float), #1-1腔体真空压力（Pa_Float）
LD TR0
@LD H26.00  ; #1-1电池泄漏
@OR T1920  ; #1-1电池抽真空阈值到达延时（测试）
ANDLD
@MOVF(469) D902 D218  ; #1-1电池实际真空值(Float), #1-1电池真空压力（Pa_Float）
LD TR0
LD D1066.10  ; #1腔体机构开腔体氦检阀/延时关腔体抽气阀（自动步）
OR D1070.09  ; #1腔体机构开腔体氦检阀/延时关腔体抽气阀（自动单检步）
ANDLD
ANDNOT H26.00  ; #1-1电池泄漏
ANDNOT H26.02  ; #1-1电池注氦超时
@AND T1904  ; #1-1腔体氦检时间（测试）
@MOVF(469) D990 D202  ; 实时漏率（Pa.m3/s_Float）, #1-1腔体测试漏率（Pa.m3/s_Float）
@MOVF(469) D992 D204  ; 实时检漏口压力（Pa_Float）, #1-1腔体测试检漏口压力（Pa_Float）
LD TR0
AND D1075.00  ; #1腔体机构腔体氦检阀仪真空阀打开/延时关腔体抽气阀（清氦步）
@AND T1904  ; #1-1腔体氦检时间（测试）
MOVF(469) D990 D258  ; 实时漏率（Pa.m3/s_Float）, #1-1清氦泄漏率（清氦）

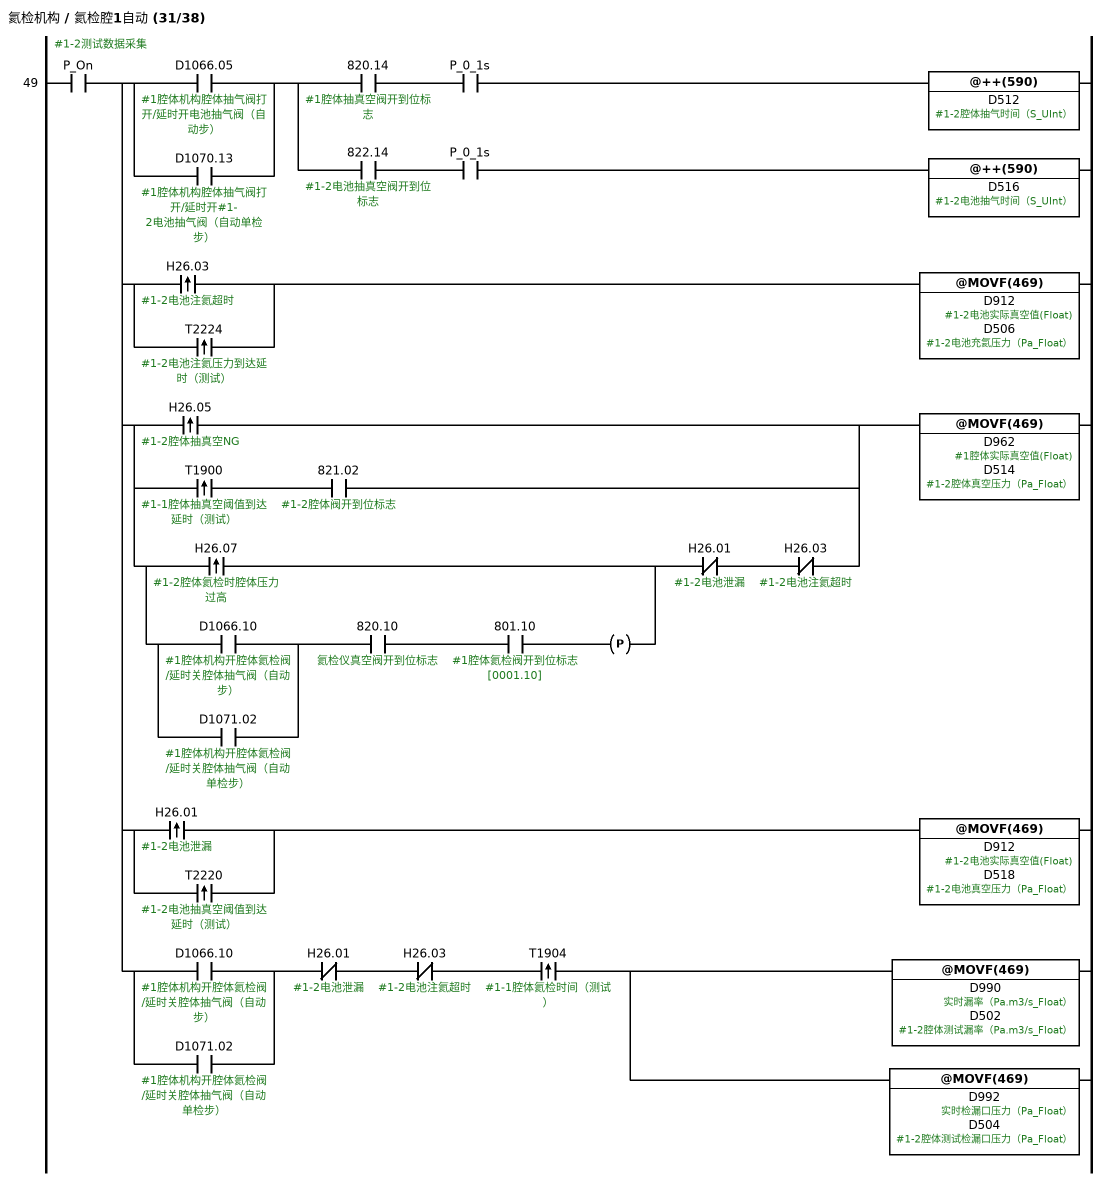
; rung 49: #1-2测试数据采集
LD P_On
OUT TR0
LD D1066.05  ; #1腔体机构腔体抽气阀打开/延时开电池抽气阀（自动步）
OR D1070.13  ; #1腔体机构腔体抽气阀打开/延时开#1-2电池抽气阀（自动单检步）
ANDLD
OUT TR1
AND 820.14  ; #1腔体抽真空阀开到位标志
AND P_0_1s
@++(590) D512  ; #1-2腔体抽气时间（S_UInt）
LD TR1
AND 822.14  ; #1-2电池抽真空阀开到位标志
AND P_0_1s
@++(590) D516  ; #1-2电池抽气时间（S_UInt）
LD TR0
@LD H26.03  ; #1-2电池注氦超时
@OR T2224  ; #1-2电池注氦压力到达延时（测试）
ANDLD
@MOVF(469) D912 D506  ; #1-2电池实际真空值(Float), #1-2电池充氦压力（Pa_Float）
LD TR0
@LD H26.05  ; #1-2腔体抽真空NG
@LD T1900  ; #1-1腔体抽真空阈值到达延时（测试）
AND 821.02  ; #1-2腔体阀开到位标志
ORLD
@LD H26.07  ; #1-2腔体氦检时腔体压力过高
LD D1066.10  ; #1腔体机构开腔体氦检阀/延时关腔体抽气阀（自动步）
OR D1071.02  ; #1腔体机构开腔体氦检阀/延时关腔体抽气阀（自动单检步）
AND 820.10  ; 氦检仪真空阀开到位标志
AND 801.10  ; #1腔体氦检阀开到位标志[0001.10]
UP(521)
ORLD
ANDNOT H26.01  ; #1-2电池泄漏
ANDNOT H26.03  ; #1-2电池注氦超时
ORLD
ANDLD
@MOVF(469) D962 D514  ; #1腔体实际真空值(Float), #1-2腔体真空压力（Pa_Float）
LD TR0
@LD H26.01  ; #1-2电池泄漏
@OR T2220  ; #1-2电池抽真空阈值到达延时（测试）
ANDLD
@MOVF(469) D912 D518  ; #1-2电池实际真空值(Float), #1-2电池真空压力（Pa_Float）
LD TR0
LD D1066.10  ; #1腔体机构开腔体氦检阀/延时关腔体抽气阀（自动步）
OR D1071.02  ; #1腔体机构开腔体氦检阀/延时关腔体抽气阀（自动单检步）
ANDLD
ANDNOT H26.01  ; #1-2电池泄漏
ANDNOT H26.03  ; #1-2电池注氦超时
@AND T1904  ; #1-1腔体氦检时间（测试）
@MOVF(469) D990 D502  ; 实时漏率（Pa.m3/s_Float）, #1-2腔体测试漏率（Pa.m3/s_Float）
@MOVF(469) D992 D504  ; 实时检漏口压力（Pa_Float）, #1-2腔体测试检漏口压力（Pa_Float）

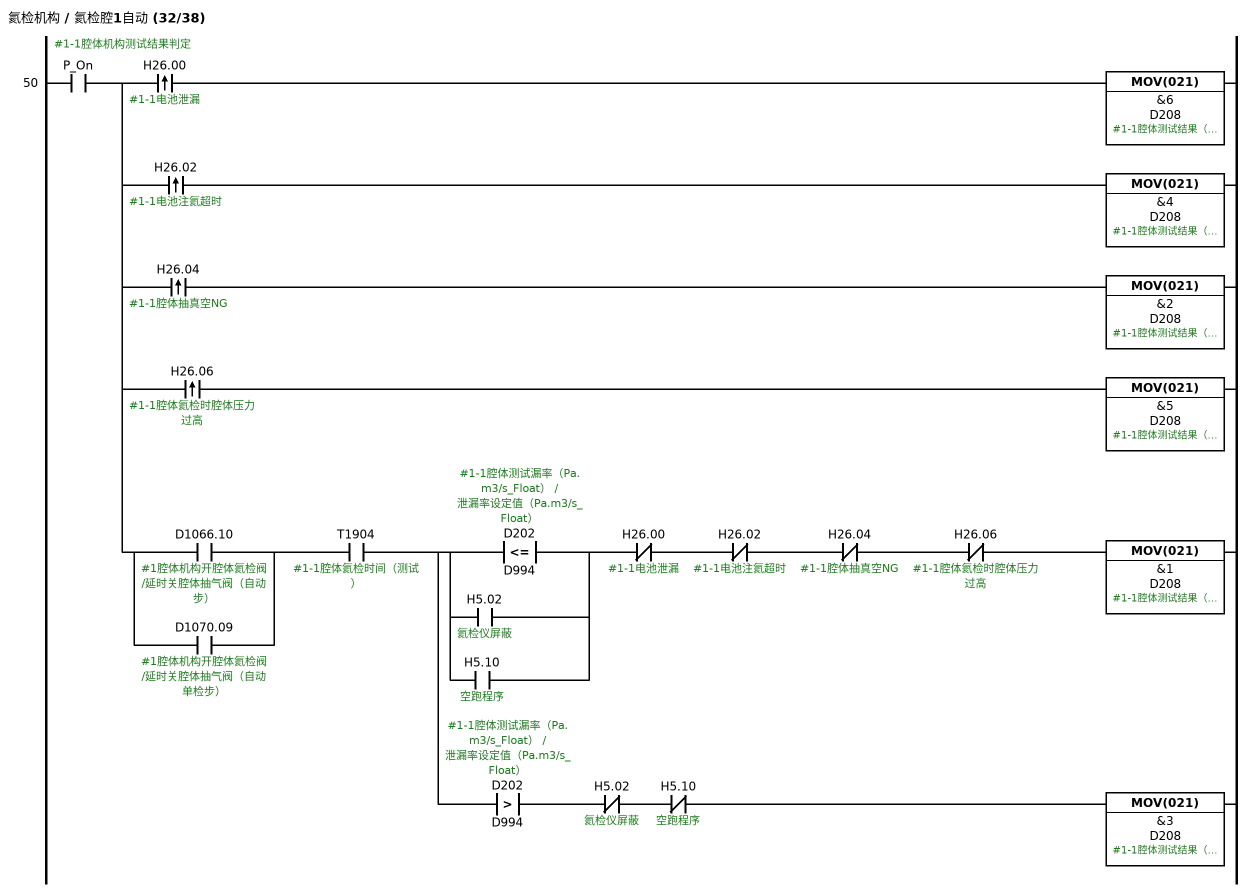
; rung 50: #1-1腔体机构测试结果判定
LD P_On
OUT TR0
@AND H26.00  ; #1-1电池泄漏
MOV(021) &6 D208  ; #1-1腔体测试结果（1 OK，2腔体泄漏，3气密NG，4注氦超时，5氦检异常，6电池泄漏）
LD TR0
@AND H26.02  ; #1-1电池注氦超时
MOV(021) &4 D208  ; #1-1腔体测试结果（1 OK，2腔体泄漏，3气密NG，4注氦超时，5氦检异常，6电池泄漏）
LD TR0
@AND H26.04  ; #1-1腔体抽真空NG
MOV(021) &2 D208  ; #1-1腔体测试结果（1 OK，2腔体泄漏，3气密NG，4注氦超时，5氦检异常，6电池泄漏）
LD TR0
@AND H26.06  ; #1-1腔体氦检时腔体压力过高
MOV(021) &5 D208  ; #1-1腔体测试结果（1 OK，2腔体泄漏，3气密NG，4注氦超时，5氦检异常，6电池泄漏）
LD TR0
LD D1066.10  ; #1腔体机构开腔体氦检阀/延时关腔体抽气阀（自动步）
OR D1070.09  ; #1腔体机构开腔体氦检阀/延时关腔体抽气阀（自动单检步）
ANDLD
AND T1904  ; #1-1腔体氦检时间（测试）
OUT TR0
LD<=F(332) D202 D994  ; #1-1腔体测试漏率（Pa.m3/s_Float）, 泄漏率设定值（Pa.m3/s_Float）
OR H5.02  ; 氦检仪屏蔽
OR H5.10  ; 空跑程序
ANDLD
ANDNOT H26.00  ; #1-1电池泄漏
ANDNOT H26.02  ; #1-1电池注氦超时
ANDNOT H26.04  ; #1-1腔体抽真空NG
ANDNOT H26.06  ; #1-1腔体氦检时腔体压力过高
MOV(021) &1 D208  ; #1-1腔体测试结果（1 OK，2腔体泄漏，3气密NG，4注氦超时，5氦检异常，6电池泄漏）
LD TR0
AND>F(333) D202 D994  ; #1-1腔体测试漏率（Pa.m3/s_Float）, 泄漏率设定值（Pa.m3/s_Float）
ANDNOT H5.02  ; 氦检仪屏蔽
ANDNOT H5.10  ; 空跑程序
MOV(021) &3 D208  ; #1-1腔体测试结果（1 OK，2腔体泄漏，3气密NG，4注氦超时，5氦检异常，6电池泄漏）

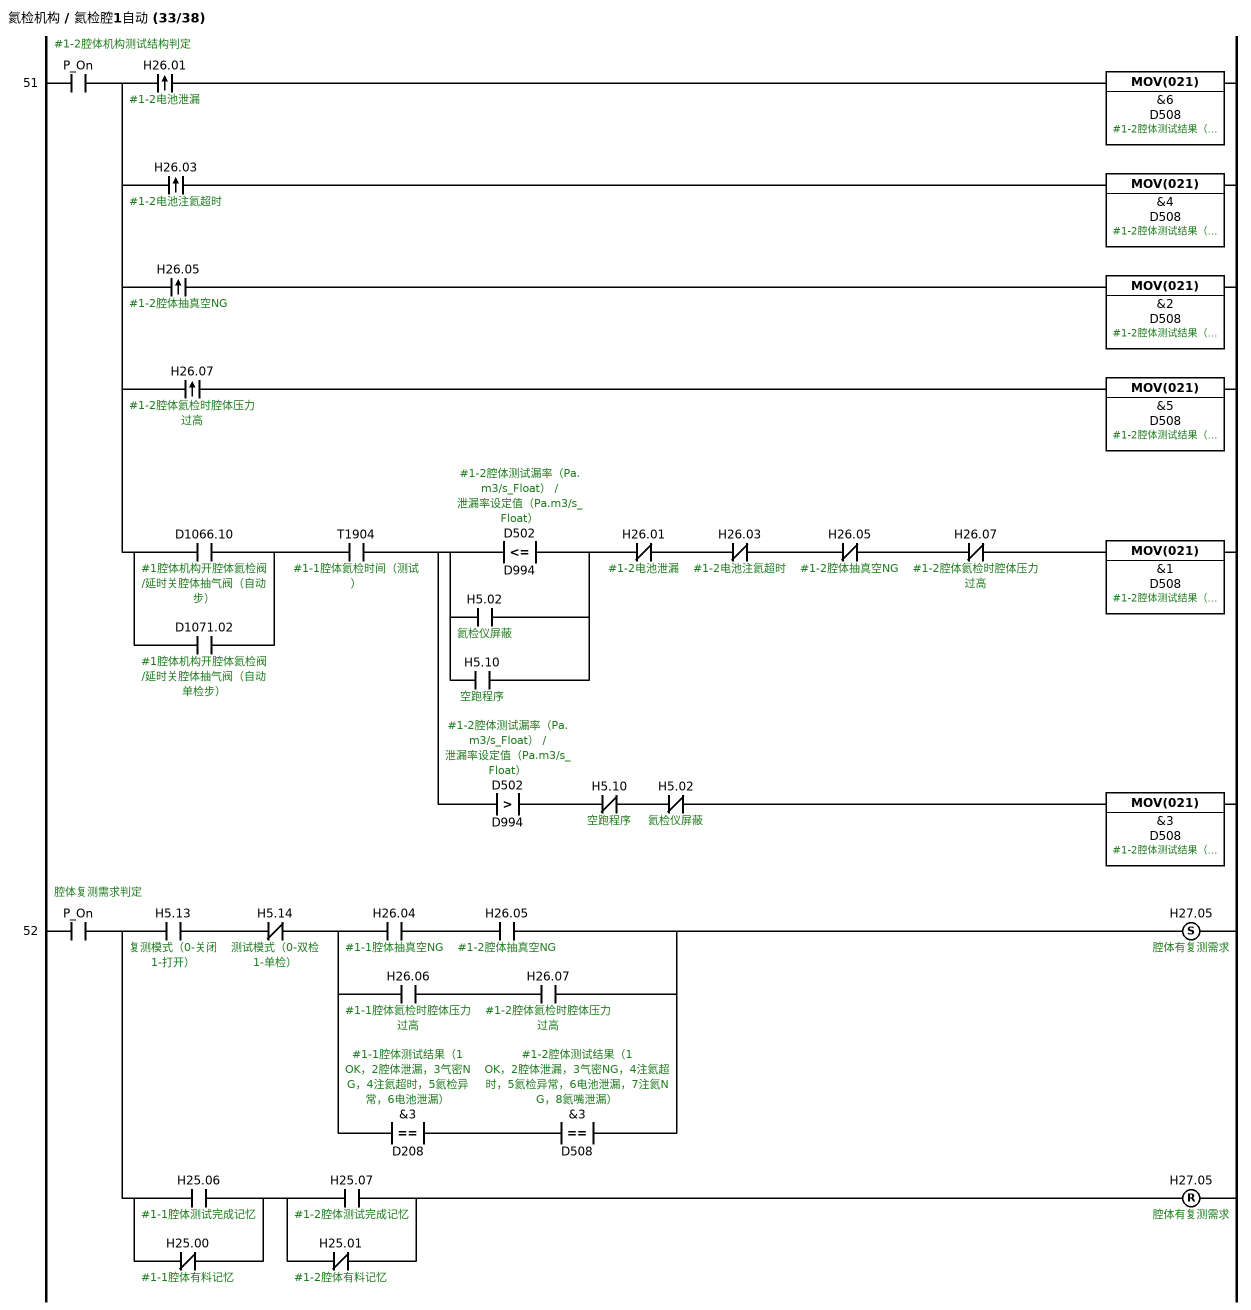
; rung 51: #1-2腔体机构测试结构判定
LD P_On
OUT TR0
@AND H26.01  ; #1-2电池泄漏
MOV(021) &6 D508  ; #1-2腔体测试结果（1 OK，2腔体泄漏，3气密NG，4注氦超时，5氦检异常，6电池泄漏，7注氦NG，8氦嘴泄漏）
LD TR0
@AND H26.03  ; #1-2电池注氦超时
MOV(021) &4 D508  ; #1-2腔体测试结果（1 OK，2腔体泄漏，3气密NG，4注氦超时，5氦检异常，6电池泄漏，7注氦NG，8氦嘴泄漏）
LD TR0
@AND H26.05  ; #1-2腔体抽真空NG
MOV(021) &2 D508  ; #1-2腔体测试结果（1 OK，2腔体泄漏，3气密NG，4注氦超时，5氦检异常，6电池泄漏，7注氦NG，8氦嘴泄漏）
LD TR0
@AND H26.07  ; #1-2腔体氦检时腔体压力过高
MOV(021) &5 D508  ; #1-2腔体测试结果（1 OK，2腔体泄漏，3气密NG，4注氦超时，5氦检异常，6电池泄漏，7注氦NG，8氦嘴泄漏）
LD TR0
LD D1066.10  ; #1腔体机构开腔体氦检阀/延时关腔体抽气阀（自动步）
OR D1071.02  ; #1腔体机构开腔体氦检阀/延时关腔体抽气阀（自动单检步）
ANDLD
AND T1904  ; #1-1腔体氦检时间（测试）
OUT TR0
LD<=F(332) D502 D994  ; #1-2腔体测试漏率（Pa.m3/s_Float）, 泄漏率设定值（Pa.m3/s_Float）
OR H5.02  ; 氦检仪屏蔽
OR H5.10  ; 空跑程序
ANDLD
ANDNOT H26.01  ; #1-2电池泄漏
ANDNOT H26.03  ; #1-2电池注氦超时
ANDNOT H26.05  ; #1-2腔体抽真空NG
ANDNOT H26.07  ; #1-2腔体氦检时腔体压力过高
MOV(021) &1 D508  ; #1-2腔体测试结果（1 OK，2腔体泄漏，3气密NG，4注氦超时，5氦检异常，6电池泄漏，7注氦NG，8氦嘴泄漏）
LD TR0
AND>F(333) D502 D994  ; #1-2腔体测试漏率（Pa.m3/s_Float）, 泄漏率设定值（Pa.m3/s_Float）
ANDNOT H5.10  ; 空跑程序
ANDNOT H5.02  ; 氦检仪屏蔽
MOV(021) &3 D508  ; #1-2腔体测试结果（1 OK，2腔体泄漏，3气密NG，4注氦超时，5氦检异常，6电池泄漏，7注氦NG，8氦嘴泄漏）
; rung 52: 腔体复测需求判定
LD P_On
OUT TR0
AND H5.13  ; 复测模式（0-关闭 1-打开）
ANDNOT H5.14  ; 测试模式（0-双检 1-单检）
LD H26.04  ; #1-1腔体抽真空NG
AND H26.05  ; #1-2腔体抽真空NG
LD H26.06  ; #1-1腔体氦检时腔体压力过高
AND H26.07  ; #1-2腔体氦检时腔体压力过高
ORLD
LD=(300) &3 D208  ; #1-1腔体测试结果（1 OK，2腔体泄漏，3气密NG，4注氦超时，5氦检异常，6电池泄漏）
AND=(300) &3 D508  ; #1-2腔体测试结果（1 OK，2腔体泄漏，3气密NG，4注氦超时，5氦检异常，6电池泄漏，7注氦NG，8氦嘴泄漏）
ORLD
ANDLD
SET H27.05  ; 腔体有复测需求
LD TR0
LD H25.06  ; #1-1腔体测试完成记忆
ORNOT H25.00  ; #1-1腔体有料记忆
ANDLD
LD H25.07  ; #1-2腔体测试完成记忆
ORNOT H25.01  ; #1-2腔体有料记忆
ANDLD
RSET H27.05  ; 腔体有复测需求

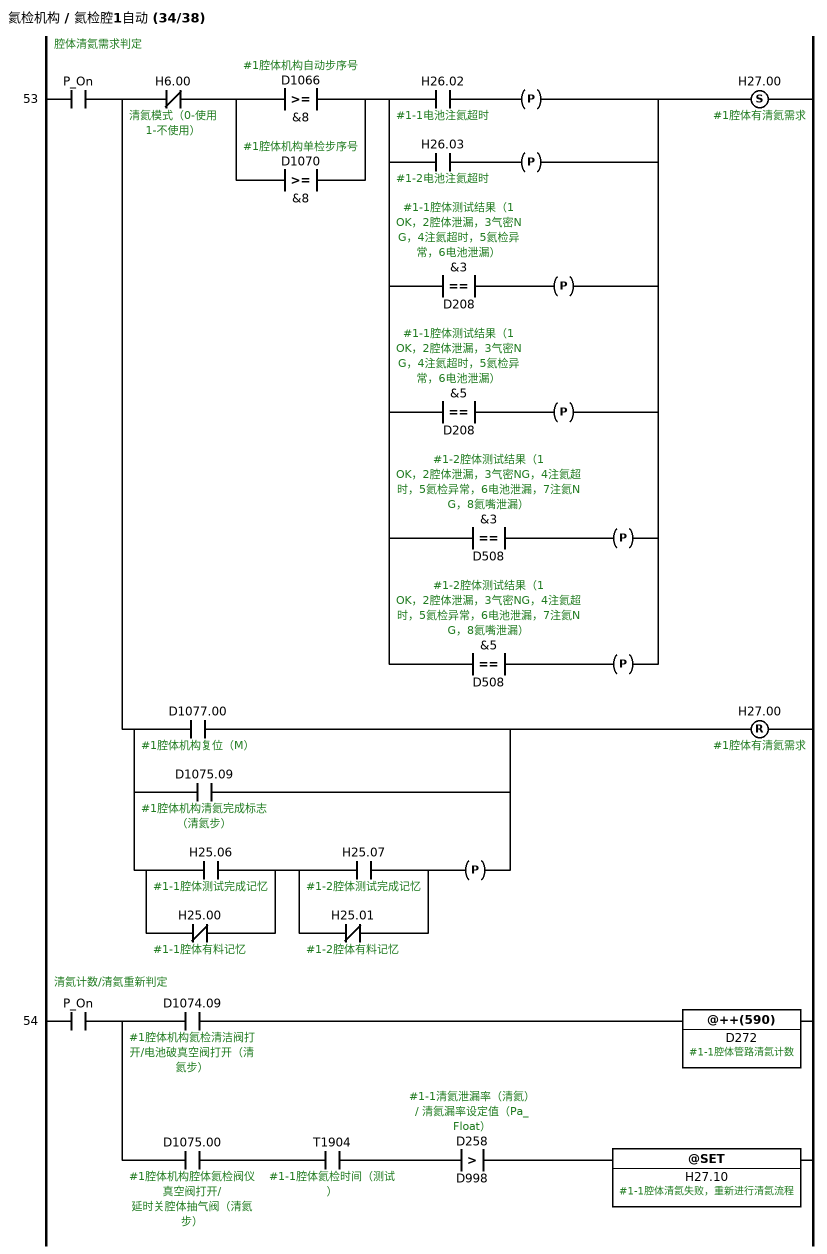
; rung 53: 腔体清氦需求判定
LD P_On
OUT TR0
ANDNOT H6.00  ; 清氦模式（0-使用 1-不使用）
LD>=L(326) D1066 &8  ; #1腔体机构自动步序号
OR>=L(326) D1070 &8  ; #1腔体机构单检步序号
ANDLD
LD H26.02  ; #1-1电池注氦超时
UP(521)
LD H26.03  ; #1-2电池注氦超时
UP(521)
ORLD
LD=(300) &3 D208  ; #1-1腔体测试结果（1 OK，2腔体泄漏，3气密NG，4注氦超时，5氦检异常，6电池泄漏）
UP(521)
ORLD
LD=(300) &5 D208  ; #1-1腔体测试结果（1 OK，2腔体泄漏，3气密NG，4注氦超时，5氦检异常，6电池泄漏）
UP(521)
ORLD
LD=(300) &3 D508  ; #1-2腔体测试结果（1 OK，2腔体泄漏，3气密NG，4注氦超时，5氦检异常，6电池泄漏，7注氦NG，8氦嘴泄漏）
UP(521)
ORLD
LD=(300) &5 D508  ; #1-2腔体测试结果（1 OK，2腔体泄漏，3气密NG，4注氦超时，5氦检异常，6电池泄漏，7注氦NG，8氦嘴泄漏）
UP(521)
ORLD
ANDLD
SET H27.00  ; #1腔体有清氦需求
LD TR0
LD D1077.00  ; #1腔体机构复位（M）
OR D1075.09  ; #1腔体机构清氦完成标志（清氦步）
LD H25.06  ; #1-1腔体测试完成记忆
ORNOT H25.00  ; #1-1腔体有料记忆
LD H25.07  ; #1-2腔体测试完成记忆
ORNOT H25.01  ; #1-2腔体有料记忆
ANDLD
UP(521)
ORLD
ANDLD
RSET H27.00  ; #1腔体有清氦需求
; rung 54: 清氦计数/清氦重新判定
LD P_On
OUT TR0
AND D1074.09  ; #1腔体机构氦检清洁阀打开/电池破真空阀打开（清氦步）
@++(590) D272  ; #1-1腔体管路清氦计数
LD TR0
AND D1075.00  ; #1腔体机构腔体氦检阀仪真空阀打开/延时关腔体抽气阀（清氦步）
AND T1904  ; #1-1腔体氦检时间（测试）
AND>F(333) D258 D998  ; #1-1清氦泄漏率（清氦）, 清氦漏率设定值（Pa_Float）
@SET H27.10  ; #1-1腔体清氦失败，重新进行清氦流程

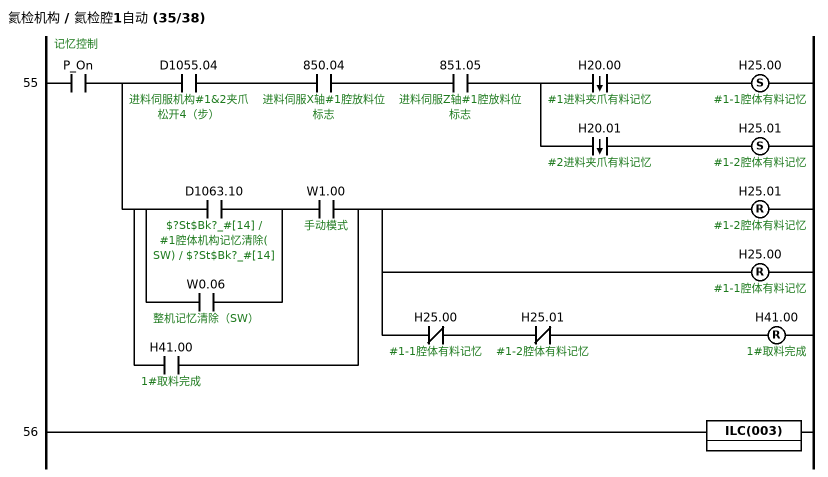
; rung 55: 记忆控制
LD P_On
OUT TR0
AND D1055.04  ; 进料伺服机构#1&2夹爪松开4（步）
AND 850.04  ; 进料伺服X轴#1腔放料位标志
AND 851.05  ; 进料伺服Z轴#1腔放料位标志
OUT TR1
%AND H20.00  ; #1进料夹爪有料记忆
SET H25.00  ; #1-1腔体有料记忆
LD TR1
%AND H20.01  ; #2进料夹爪有料记忆
SET H25.01  ; #1-2腔体有料记忆
LD TR0
LD D1063.10  ; $?St$Bk?_#[14] / #1腔体机构记忆清除(SW) / $?St$Bk?_#[14]
OR W0.06  ; 整机记忆清除（SW）
AND W1.00  ; 手动模式
OR H41.00  ; 1#取料完成
ANDLD
RSET H25.01  ; #1-2腔体有料记忆
RSET H25.00  ; #1-1腔体有料记忆
ANDNOT H25.00  ; #1-1腔体有料记忆
ANDNOT H25.01  ; #1-2腔体有料记忆
RSET H41.00  ; 1#取料完成
; rung 56
ILC(003)

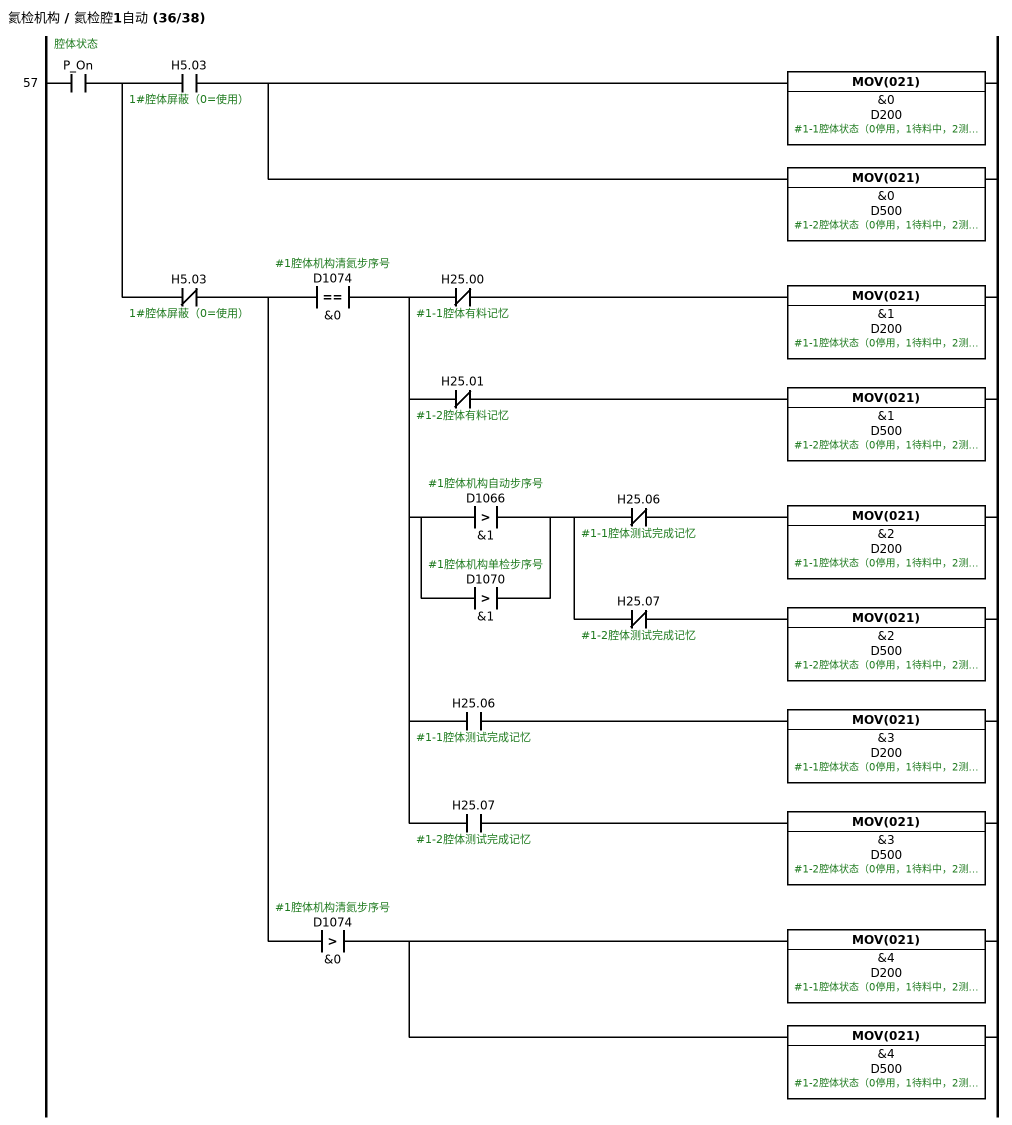
; rung 57: 腔体状态
LD P_On
OUT TR0
AND H5.03  ; 1#腔体屏蔽（0=使用）
MOV(021) &0 D200  ; #1-1腔体状态（0停用，1待料中，2测试中，3测试完成，4-清氦中）
MOV(021) &0 D500  ; #1-2腔体状态（0停用，1待料中，2测试中，3测试完成，4-清氦中）
LD TR0
ANDNOT H5.03  ; 1#腔体屏蔽（0=使用）
OUT TR0
AND=L(301) D1074 &0  ; #1腔体机构清氦步序号
OUT TR1
ANDNOT H25.00  ; #1-1腔体有料记忆
MOV(021) &1 D200  ; #1-1腔体状态（0停用，1待料中，2测试中，3测试完成，4-清氦中）
LD TR1
ANDNOT H25.01  ; #1-2腔体有料记忆
MOV(021) &1 D500  ; #1-2腔体状态（0停用，1待料中，2测试中，3测试完成，4-清氦中）
LD TR1
LD>L(321) D1066 &1  ; #1腔体机构自动步序号
OR>L(321) D1070 &1  ; #1腔体机构单检步序号
ANDLD
OUT TR2
ANDNOT H25.06  ; #1-1腔体测试完成记忆
MOV(021) &2 D200  ; #1-1腔体状态（0停用，1待料中，2测试中，3测试完成，4-清氦中）
LD TR2
ANDNOT H25.07  ; #1-2腔体测试完成记忆
MOV(021) &2 D500  ; #1-2腔体状态（0停用，1待料中，2测试中，3测试完成，4-清氦中）
LD TR1
AND H25.06  ; #1-1腔体测试完成记忆
MOV(021) &3 D200  ; #1-1腔体状态（0停用，1待料中，2测试中，3测试完成，4-清氦中）
LD TR1
AND H25.07  ; #1-2腔体测试完成记忆
MOV(021) &3 D500  ; #1-2腔体状态（0停用，1待料中，2测试中，3测试完成，4-清氦中）
LD TR0
AND>L(321) D1074 &0  ; #1腔体机构清氦步序号
MOV(021) &4 D200  ; #1-1腔体状态（0停用，1待料中，2测试中，3测试完成，4-清氦中）
MOV(021) &4 D500  ; #1-2腔体状态（0停用，1待料中，2测试中，3测试完成，4-清氦中）

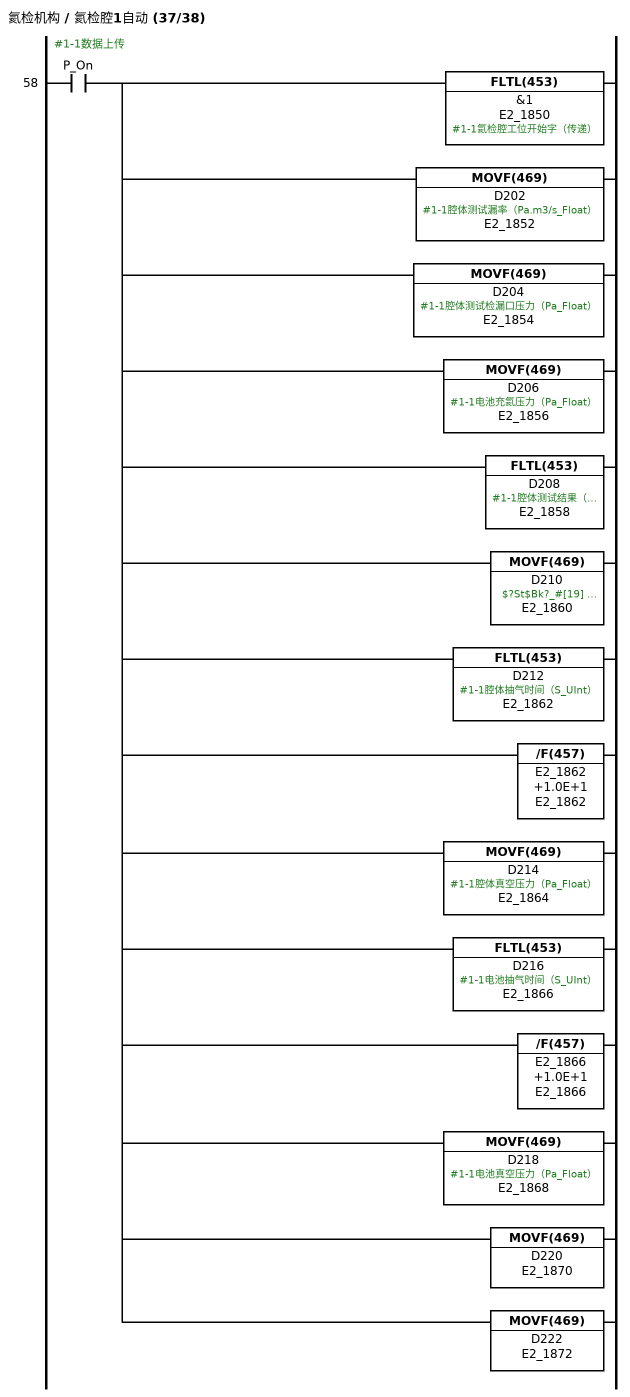
; rung 58: #1-1数据上传
LD P_On
FLTL(453) &1 E2_1850  ; #1-1氦检腔工位开始字（传递）
MOVF(469) D202 E2_1852  ; #1-1腔体测试漏率（Pa.m3/s_Float）
MOVF(469) D204 E2_1854  ; #1-1腔体测试检漏口压力（Pa_Float）
MOVF(469) D206 E2_1856  ; #1-1电池充氦压力（Pa_Float）
FLTL(453) D208 E2_1858  ; #1-1腔体测试结果（1 OK，2腔体泄漏，3气密NG，4注氦超时，5氦检异常，6电池泄漏）
MOVF(469) D210 E2_1860  ; $?St$Bk?_#[19] / #1-1充氦嘴压力（Pa_Float） / #1-1充氦嘴压力（Pa_Float） / #1-1充氦嘴压力（Pa_Float）$?St$Bk?_#[19]
FLTL(453) D212 E2_1862  ; #1-1腔体抽气时间（S_UInt）
/F(457) E2_1862 +1.0E+1 E2_1862
MOVF(469) D214 E2_1864  ; #1-1腔体真空压力（Pa_Float）
FLTL(453) D216 E2_1866  ; #1-1电池抽气时间（S_UInt）
/F(457) E2_1866 +1.0E+1 E2_1866
MOVF(469) D218 E2_1868  ; #1-1电池真空压力（Pa_Float）
MOVF(469) D220 E2_1870
MOVF(469) D222 E2_1872

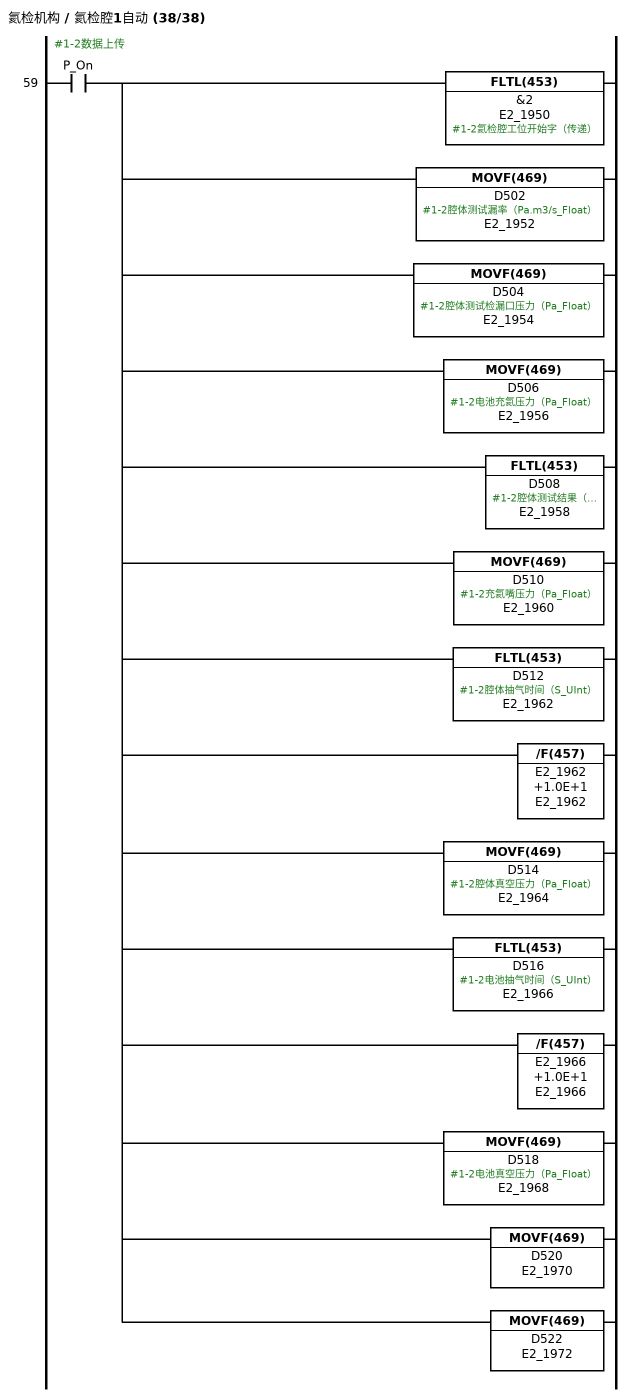
; rung 59: #1-2数据上传
LD P_On
FLTL(453) &2 E2_1950  ; #1-2氦检腔工位开始字（传递）
MOVF(469) D502 E2_1952  ; #1-2腔体测试漏率（Pa.m3/s_Float）
MOVF(469) D504 E2_1954  ; #1-2腔体测试检漏口压力（Pa_Float）
MOVF(469) D506 E2_1956  ; #1-2电池充氦压力（Pa_Float）
FLTL(453) D508 E2_1958  ; #1-2腔体测试结果（1 OK，2腔体泄漏，3气密NG，4注氦超时，5氦检异常，6电池泄漏，7注氦NG，8氦嘴泄漏）
MOVF(469) D510 E2_1960  ; #1-2充氦嘴压力（Pa_Float）
FLTL(453) D512 E2_1962  ; #1-2腔体抽气时间（S_UInt）
/F(457) E2_1962 +1.0E+1 E2_1962
MOVF(469) D514 E2_1964  ; #1-2腔体真空压力（Pa_Float）
FLTL(453) D516 E2_1966  ; #1-2电池抽气时间（S_UInt）
/F(457) E2_1966 +1.0E+1 E2_1966
MOVF(469) D518 E2_1968  ; #1-2电池真空压力（Pa_Float）
MOVF(469) D520 E2_1970
MOVF(469) D522 E2_1972

### Section 氦检腔2自动

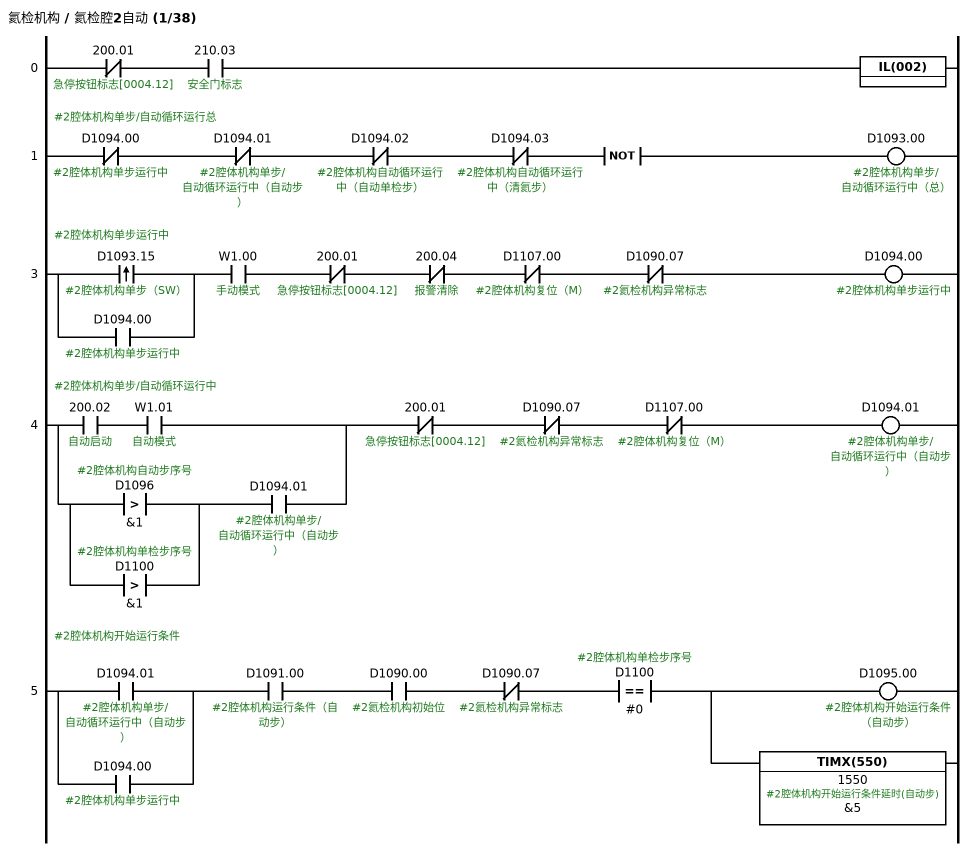
; rung 0
LDNOT 200.01  ; 急停按钮标志[0004.12]
AND 210.03  ; 安全门标志
IL(002)
; rung 1: #2腔体机构单步/自动循环运行总
LDNOT D1094.00  ; #2腔体机构单步运行中
ANDNOT D1094.01  ; #2腔体机构单步/自动循环运行中（自动步）
ANDNOT D1094.02  ; #2腔体机构自动循环运行中（自动单检步）
ANDNOT D1094.03  ; #2腔体机构自动循环运行中（清氦步）
NOT(520)
OUT D1093.00  ; #2腔体机构单步/自动循环运行中（总）
; rung 2: ******************************* / 自动双检步序 / *******************************
; rung 3: #2腔体机构单步运行中
@LD D1093.15  ; #2腔体机构单步（SW）
OR D1094.00  ; #2腔体机构单步运行中
AND W1.00  ; 手动模式
ANDNOT 200.01  ; 急停按钮标志[0004.12]
ANDNOT 200.04  ; 报警清除
ANDNOT D1107.00  ; #2腔体机构复位（M）
ANDNOT D1090.07  ; #2氦检机构异常标志
OUT D1094.00  ; #2腔体机构单步运行中
; rung 4: #2腔体机构单步/自动循环运行中
LD 200.02  ; 自动启动
AND W1.01  ; 自动模式
LD>L(321) D1096 &1  ; #2腔体机构自动步序号
OR>L(321) D1100 &1  ; #2腔体机构单检步序号
AND D1094.01  ; #2腔体机构单步/自动循环运行中（自动步）
ORLD
ANDNOT 200.01  ; 急停按钮标志[0004.12]
ANDNOT D1090.07  ; #2氦检机构异常标志
ANDNOT D1107.00  ; #2腔体机构复位（M）
OUT D1094.01  ; #2腔体机构单步/自动循环运行中（自动步）
; rung 5: #2腔体机构开始运行条件
LD D1094.01  ; #2腔体机构单步/自动循环运行中（自动步）
OR D1094.00  ; #2腔体机构单步运行中
AND D1091.00  ; #2腔体机构运行条件（自动步）
AND D1090.00  ; #2氦检机构初始位
ANDNOT D1090.07  ; #2氦检机构异常标志
AND=L(301) D1100 #0  ; #2腔体机构单检步序号
OUT D1095.00  ; #2腔体机构开始运行条件（自动步）
TIMX(550) 1550 &5  ; #2腔体机构开始运行条件延时(自动步)

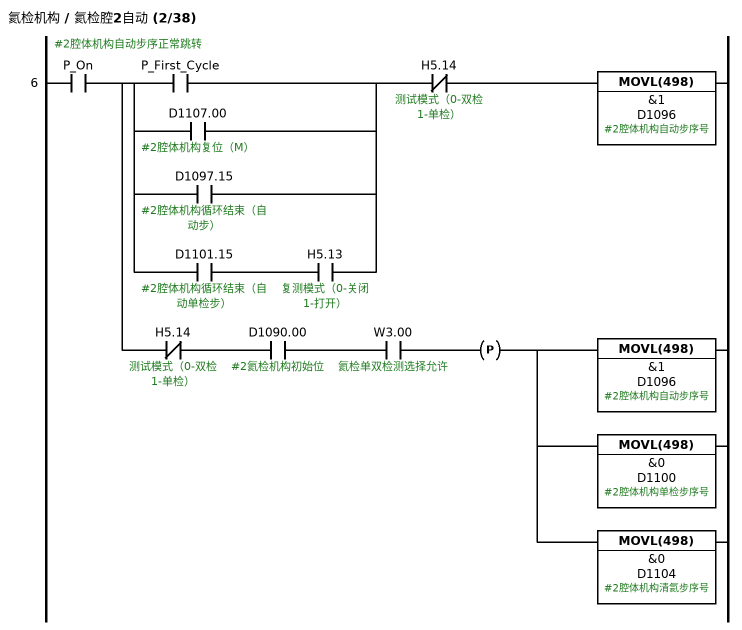
; rung 6: #2腔体机构自动步序正常跳转
LD P_On
OUT TR0
LD P_First_Cycle
OR D1107.00  ; #2腔体机构复位（M）
OR D1097.15  ; #2腔体机构循环结束（自动步）
LD D1101.15  ; #2腔体机构循环结束（自动单检步）
AND H5.13  ; 复测模式（0-关闭 1-打开）
ORLD
ANDLD
ANDNOT H5.14  ; 测试模式（0-双检 1-单检）
MOVL(498) &1 D1096  ; #2腔体机构自动步序号
LD TR0
ANDNOT H5.14  ; 测试模式（0-双检 1-单检）
AND D1090.00  ; #2氦检机构初始位
AND W3.00  ; 氦检单双检测选择允许
UP(521)
MOVL(498) &1 D1096  ; #2腔体机构自动步序号
MOVL(498) &0 D1100  ; #2腔体机构单检步序号
MOVL(498) &0 D1104  ; #2腔体机构清氦步序号

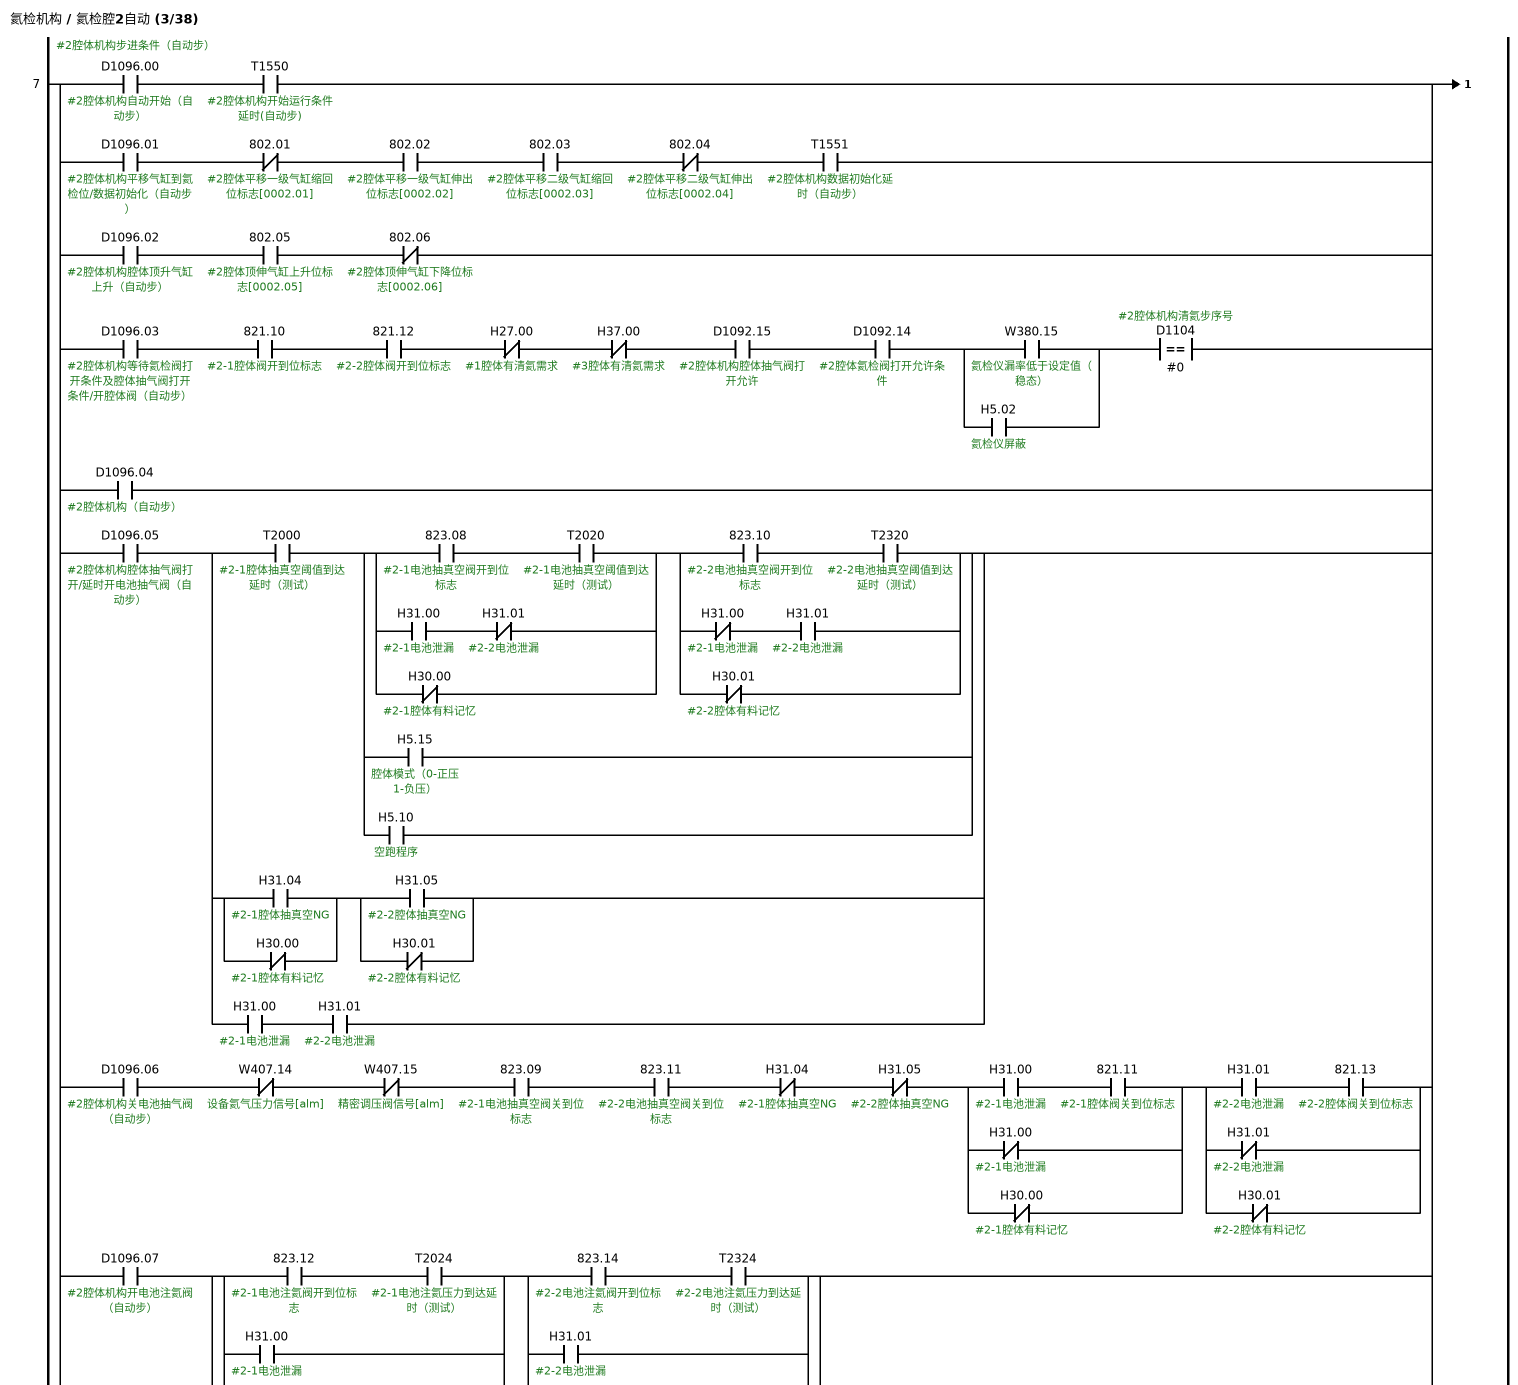

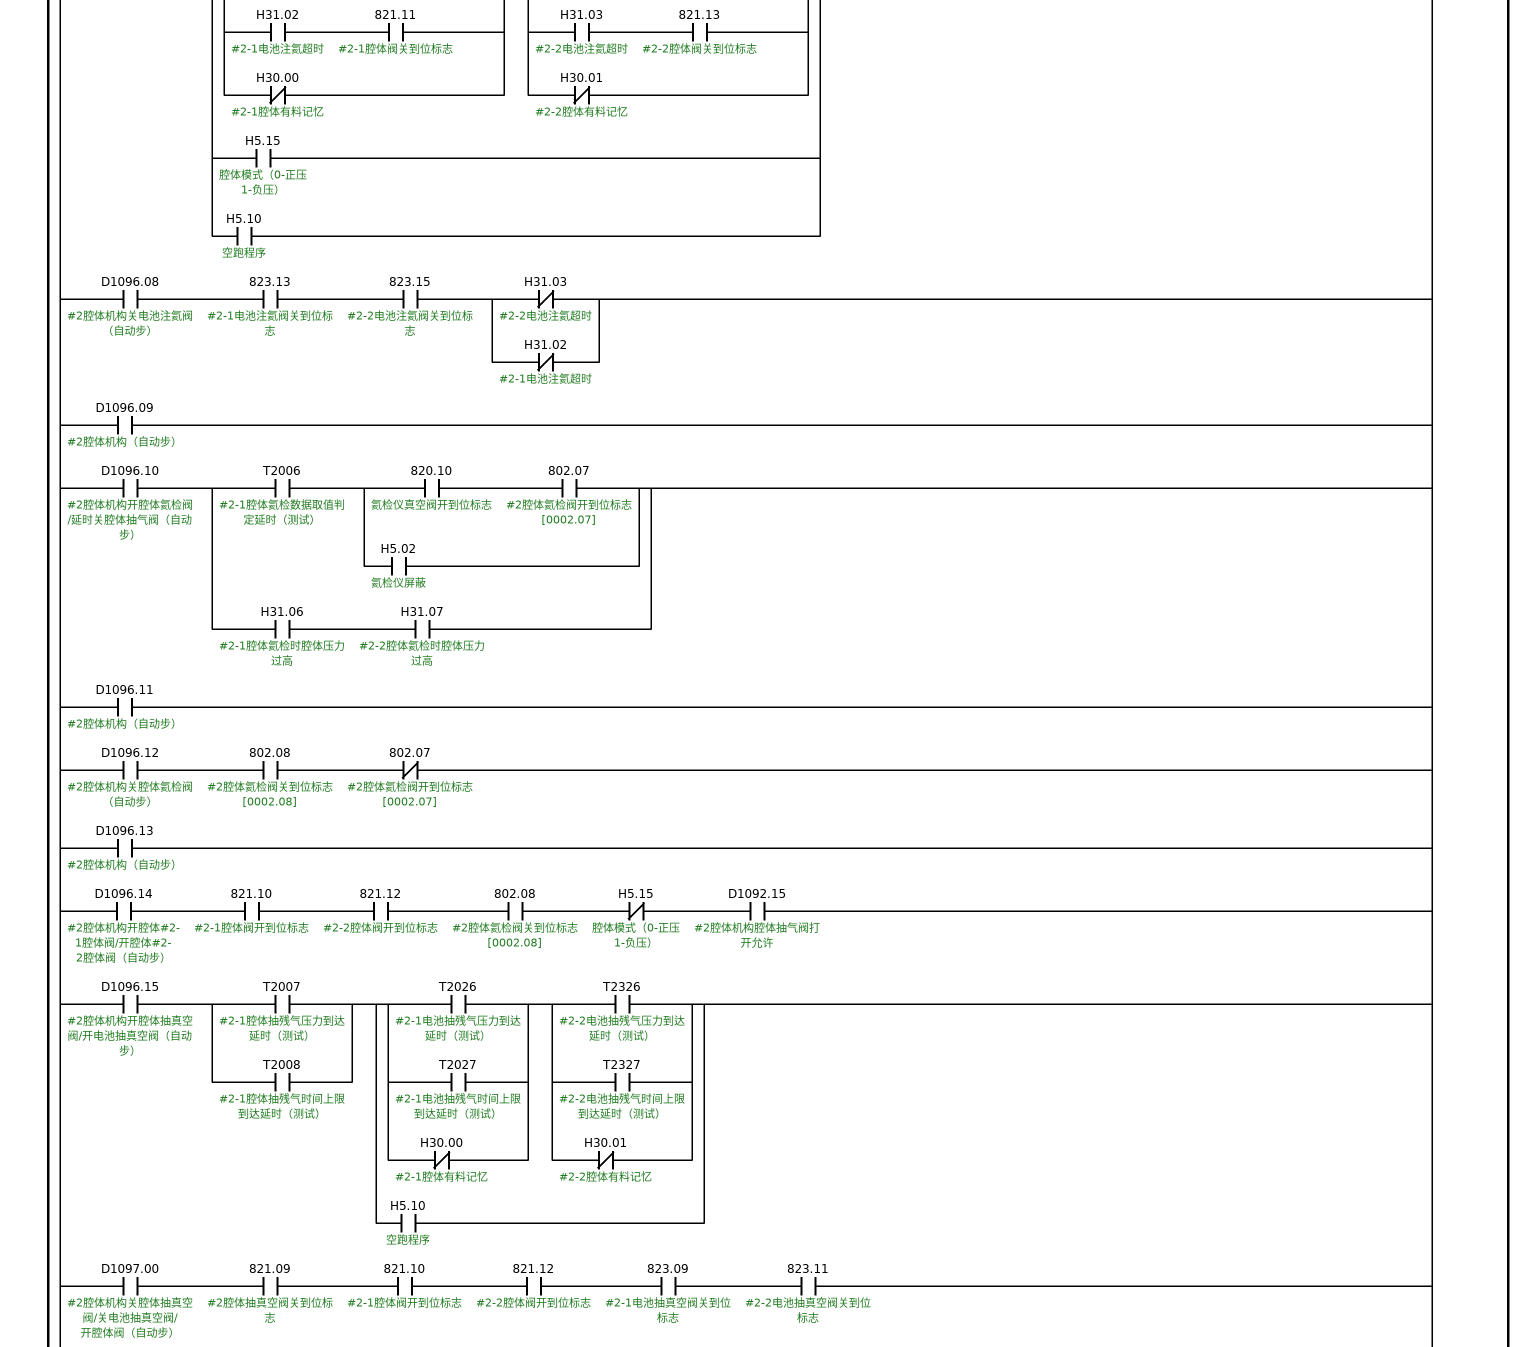

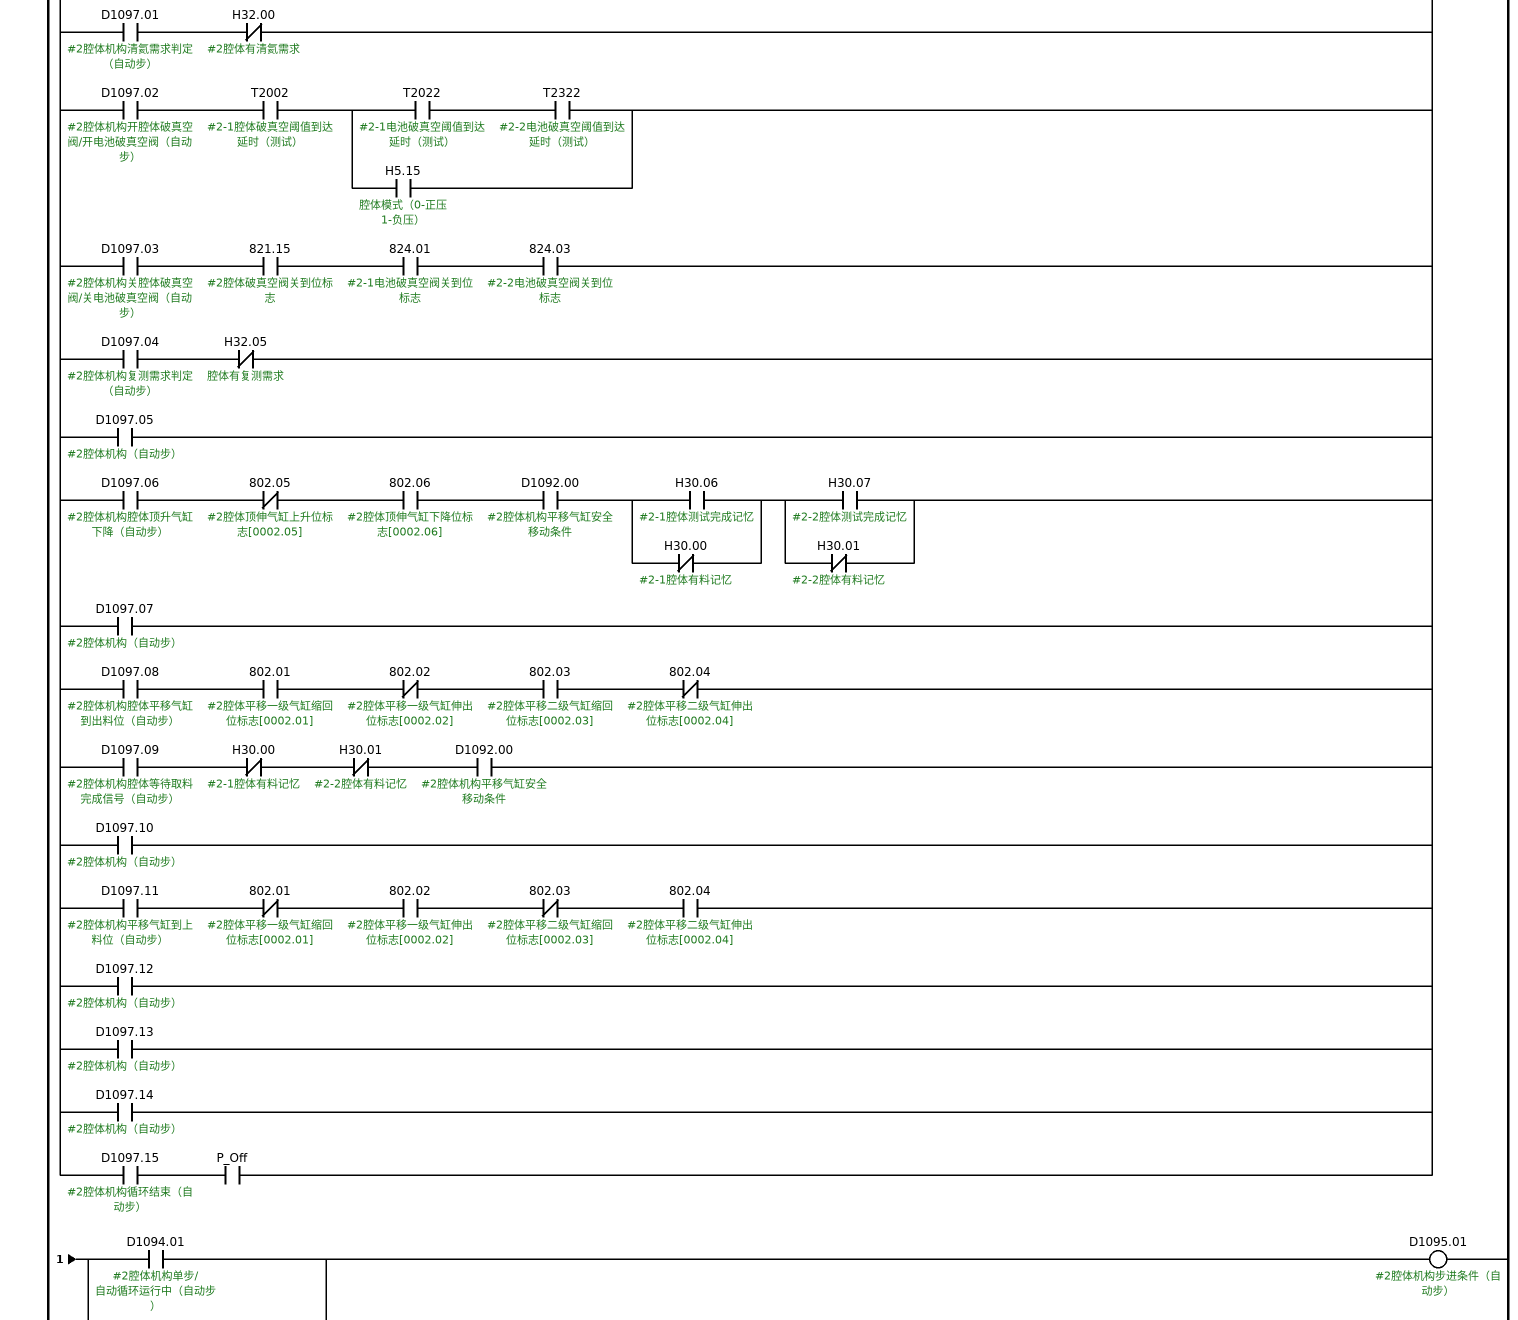

